(* PLC project Система умного дома.project, CODESYS CODESYS V3.5 SP17 Patch 3 *)
(* stored: creationDateTime 2026-04-06T20:38:17.5908527, modificationDateTime 2026-03-25T09:46:39.3897592 *)

{attribute 'qualified_only'}
{attribute 'strict'}
TYPE E_ALERT_PRIORITY : (ALERT_PRIORITY_NONE := 0, ALERT_PRIORITY_LOW := 1, ALERT_PRIORITY_MEDIUM := 2, ALERT_PRIORITY_HIGH := 3, ALERT_PRIORITY_CRITICAL := 4) BYTE;
END_TYPE

{attribute 'qualified_only'}
{attribute 'strict'}
TYPE E_Debug_Log_Level : (LOG_LEVEL_MINIMAL := 0, LOG_LEVEL_NORMAL := 1, LOG_LEVEL_VERBOSE := 2, LOG_LEVEL_DEBUG := 3) BYTE;
END_TYPE

{attribute 'qualified_only'}
{attribute 'strict'}
TYPE E_Lifetime_Device_Type : (LIFETIME_DEVICE_PUMP := 1, LIFETIME_DEVICE_FAN := 2) BYTE;
END_TYPE

{attribute 'qualified_only'}
{attribute 'strict'}
TYPE E_Outdoor_Mode : (OUTDOOR_MODE_AUTO := 0, OUTDOOR_MODE_PARTY := 1, OUTDOOR_MODE_SECURITY := 2, OUTDOOR_MODE_ECONOMY := 3, OUTDOOR_MODE_MANUAL := 4) BYTE;
END_TYPE

{attribute 'qualified_only'}
{attribute 'strict'}
TYPE E_PLC_ROLE : (ROLE_UNDEFINED := 0, ROLE_ACTIVE := 1, ROLE_STANDBY := 2, ROLE_OFFLINE := 3) USINT;
END_TYPE

{attribute 'qualified_only'}
{attribute 'strict'}
TYPE E_Rule_Action_Type : (ACTION_NONE := 0, ACTION_SET_FLOOR_HEATING := 1, ACTION_SET_LIGHTING_BASE := 2, ACTION_SET_LIGHTING_ACCENT := 3, ACTION_SET_SOCKET := 4, ACTION_SET_VENTILATION := 5, ACTION_SET_BLINDS := 6, ACTION_ACTIVATE_SCENARIO := 7, ACTION_TOGGLE_LIGHTING := 8, ACTION_TOGGLE_SOCKET := 9) BYTE;
END_TYPE

{attribute 'qualified_only'}
{attribute 'strict'}
TYPE E_Rule_Comparison : (COMP_NONE := 0, COMP_EQ := 1, COMP_GT := 2, COMP_LT := 3, COMP_GE := 4, COMP_LE := 5, COMP_IN_RANGE := 6, COMP_TRUE := 7, COMP_FALSE := 8) BYTE;
END_TYPE

(* values of E_Rule_Condition_Type: COND_AND: Логическое И (Rule Chaining); COND_OR: Логическое ИЛИ (Rule Chaining) *)

{attribute 'qualified_only'}
{attribute 'strict'}
TYPE E_Rule_Condition_Type : (COND_NONE := 0, COND_AIR_TEMP := 1, COND_FLOOR_TEMP := 2, COND_HUMIDITY := 3, COND_CO2 := 4, COND_METHANE := 5, COND_CO := 6, COND_DOOR_WINDOW := 7, COND_FLOOD := 8, COND_SMOKE := 9, COND_MOTION := 10, COND_TIME_OF_DAY := 11, COND_DAY_OF_WEEK := 12, COND_AND := 13, COND_OR := 14) BYTE;
END_TYPE

{attribute 'qualified_only'}
{attribute 'strict'}
TYPE E_SCENARIO_TYPE : (SCENARIO_NONE := 0, SCENARIO_MORNING := 1, SCENARIO_EVENING := 2, SCENARIO_AWAY := 3, SCENARIO_PARTY := 4, SCENARIO_SLEEP := 5, SCENARIO_EMERGENCY := 6, SCENARIO_PRESENCE := 7) BYTE;
END_TYPE

{attribute 'qualified_only'}
{attribute 'strict'}
TYPE E_SENSOR_TYPE : (SENSOR_TYPE_NONE := 0, SENSOR_TYPE_DOOR_WINDOW := 5, SENSOR_TYPE_GLASS_BREAK := 6, SENSOR_TYPE_FLOOD := 7, SENSOR_TYPE_SMOKE := 8, SENSOR_TYPE_GAS_METHANE := 1, SENSOR_TYPE_GAS_CO := 2, SENSOR_TYPE_TEMP_FLOOR := 3, SENSOR_TYPE_TEMP_AIR := 4) USINT;
END_TYPE

{attribute 'qualified_only'}
{attribute 'strict'}
TYPE E_Trend_Parameter_Type : (TREND_PARAM_NONE := 0, TREND_PARAM_TEMP_AIR := 1, TREND_PARAM_TEMP_FLOOR := 2, TREND_PARAM_PRESSURE := 3, TREND_PARAM_PUMP_CURRENT := 4, TREND_PARAM_GAS_METHANE := 5, TREND_PARAM_GAS_CO := 6) BYTE;
END_TYPE

{attribute 'qualified_only'}
{attribute 'strict'}
TYPE E_TwoFactor_Method : (TF_METHOD_NONE := 0, TF_METHOD_RFID := 1, TF_METHOD_TOTP := 2, TF_METHOD_BOTH := 3) BYTE;
END_TYPE

{attribute 'qualified_only'}
{attribute 'strict'}
TYPE E_Valve_Test_Result : (TEST_RESULT_NONE := 0, TEST_RESULT_PASSED := 1, TEST_RESULT_CURRENT_DEVIATION := 2, TEST_RESULT_TIME_DEVIATION := 3, TEST_RESULT_STALL := 4, TEST_RESULT_LIMIT_SWITCH_FAIL := 5, TEST_RESULT_ABORTED := 6) BYTE;
END_TYPE

(* values of E_VALVE_TYPE: VALVE_NC: Нормально-закрытый; VALVE_NO: Нормально-открытый *)

{attribute 'qualified_only'}
{attribute 'strict'}
TYPE E_VALVE_TYPE : (VALVE_NC := 1, VALVE_NO := 2) USINT;
END_TYPE

{attribute 'qualified_only'}
{attribute 'strict'}
TYPE E_VENTILATION_LOCATION : (VENT_LOCATION_NONE := 0, VENT_LOCATION_BASEMENT_GAME_ROOM := 1, VENT_LOCATION_BASEMENT_GYM := 2, VENT_LOCATION_BASEMENT_BOILER_ROOM := 3, VENT_LOCATION_BATHROOM_1F := 4, VENT_LOCATION_BATHROOM_2F := 5, VENT_LOCATION_MASTER_BATHROOM := 6, VENT_LOCATION_LAUNDRY := 7, VENT_LOCATION_KITCHEN := 8) BYTE;
END_TYPE

{attribute 'qualified_only'}
{attribute 'strict'}
TYPE E_VENTILATION_UNIT_TYPE : (VENTILATION_TYPE_NONE := 0, VENTILATION_TYPE_SUPPLY := 1, VENTILATION_TYPE_EXHAUST := 2) USINT;
END_TYPE

{attribute 'qualified_only'}
{attribute 'strict'}
TYPE E_WEATHER_COMPENSATION_METHOD : (WEATHER_COMP_NONE := 0, WEATHER_COMP_OUTDOOR_RESET := 1) USINT;
END_TYPE

{attribute 'qualified_only'}
{attribute 'strict'}
TYPE E_Zone_Access_Level : (ZONE_ACCESS_NONE := 0, ZONE_ACCESS_VIEW := 1, ZONE_ACCESS_CONTROL := 2, ZONE_ACCESS_CONFIG := 3, ZONE_ACCESS_FULL := 4) BYTE;
END_TYPE

TYPE ST_Astro_Time : STRUCT
  sunrise_ms : UDINT := 0;
  sunset_ms : UDINT := 0;
  is_daylight : BOOL := FALSE;
END_STRUCT;
END_TYPE

TYPE ST_BlackBox_Record : STRUCT
  Timestamp : UDINT;
  Gas_Methane_LEL : REAL;
  Gas_CO_PPM : REAL;
  Flood_Active : BOOL;
  Fire_Active : BOOL;
  Valve_Gas_Status : BYTE;
  Valve_Water_Status : BYTE;
  PLC_Active_ID : BYTE;
END_STRUCT;
END_TYPE

TYPE ST_Boiler_Status : STRUCT
  Active : BOOL;
  Running : BOOL;
  Error : BOOL;
  Power_Percent : REAL;
  Current_Power : REAL;
  Work_Seconds : UDINT;
  Work_Hours : REAL;
  Resource_Percent : REAL := 100;
  Last_Start : DT;
END_STRUCT;
END_TYPE

TYPE ST_Component_Maintenance : STRUCT
  Is_Faulty : BOOL;  (* Устройство неисправно *)
  Is_In_Maintenance : BOOL;  (* Выведено в ремонт вручную *)
  Fallback_Value : REAL;  (* Значение для подстановки (0-100% или температура) *)
  Use_Last_Good_Value : BOOL;  (* Использовать последнее достоверное значение *)
END_STRUCT;
END_TYPE

TYPE ST_Debug_Log_Record : STRUCT
  timestamp_ms : UDINT;
  level : BYTE;  (* E_Debug_Log_Level *)
  source_id : BYTE;
  event_code : WORD;
  value_int : UDINT;
  value_real : REAL;
  text : STRING(80);
  crc32 : DWORD;
END_STRUCT;
END_TYPE

TYPE ST_Debug_Logger_Config : STRUCT
  enabled : BOOL;
  sampling_period_ms : UDINT := 1000;
END_STRUCT;
END_TYPE

TYPE ST_Device_Health : STRUCT
  Health_Score : BYTE := 100;  (* 0..100% *)
  Total_Runtime_Hours : UDINT;
  Starts_Count : UDINT;
  Last_Start_Current : REAL;
  Avg_Start_Current : REAL;
  Maintenance_Required : BOOL;
  Warning_Message : STRING(50);
END_STRUCT;
END_TYPE

TYPE ST_DHW_Config : STRUCT
  Target_Temp : REAL := 55;
  Hysteresis : REAL := 2;
  Circulation_Schedule_Enabled : BOOL := TRUE;
  Circulation_Start : TOD := TIME_OF_DAY#6:0;
  Circulation_End : TOD := TIME_OF_DAY#23:0;
  Anti_Legionella_Enabled : BOOL := TRUE;
  Anti_Legionella_Day : UINT := 7;  (* Воскресенье *)
END_STRUCT;
END_TYPE

TYPE ST_DHW_Status : STRUCT
  Temp : REAL;
  Pressure : REAL;
  Heating_Pump_On : BOOL;
  Circ_Pump_On : BOOL;
  Error : BOOL;
  Error_ID : WORD;
END_STRUCT;
END_TYPE

TYPE ST_Flood_Config : STRUCT
  Emergency_Two_Stage_Enabled : BOOL := TRUE;  (* ТЗ 4.4 *)
  Valve_Test_Period_Days : UINT := 7;  (* ТЗ 12.2 *)
  Current_Threshold_MA : REAL := 500;  (* Порог тока для диагностики *)
END_STRUCT;
END_TYPE

TYPE ST_Flood_Global_Config : STRUCT
  valve_types : ARRAY[1..3] OF E_VALVE_TYPE := [3(E_VALVE_TYPE.VALVE_NC)];
  min_duration_ms : UDINT := 30000;
END_STRUCT;
END_TYPE

TYPE ST_FloorHeating_Circuit_Config : STRUCT
  circuit_id : BYTE := 0;
  zone : BYTE := 0;
  design_temp : REAL := 35;
  min_temp : REAL := 20;
  max_temp : REAL := 45;
  pid_kp : REAL := 2;
END_STRUCT;
END_TYPE

TYPE ST_FloorHeating_Global_Config : STRUCT
  enable_floor_heating : BOOL := TRUE;
  anti_freeze_temp : REAL := 7;
  overheat_temp : REAL := 45;
  weather_compensation_enabled : BOOL := TRUE;
  total_circuits : BYTE := 16;
END_STRUCT;
END_TYPE

TYPE ST_FloorHeating_Manifold_Config : STRUCT
  manifold_id : BYTE;
  location : STRING(30);
  nominal_flow : REAL;
  enable_pump : BOOL;
  circuits : ARRAY[1..4] OF ST_FloorHeating_Circuit_Config;
END_STRUCT;
END_TYPE

TYPE ST_Gas_Valve_Configuration : STRUCT
  valve_id : BYTE := 0;
  valve_type : E_VALVE_TYPE := E_VALVE_TYPE.VALVE_NC;
  close_time_seconds : UDINT := 10;
  open_time_seconds : UDINT := 10;
  emergency_open_allowed : BOOL := FALSE;
END_STRUCT;
END_TYPE

TYPE ST_Gateway_Command : STRUCT
  command_id : UDINT;
  timestamp_ms : UDINT;
  operator_id : STRING(10);
  command_type : BYTE;
  target_zone : BYTE;
  target_value : REAL;
  target_on_off : BOOL;
  target_scenario : E_SCENARIO_TYPE;
  target_armed : BOOL;
  crc32 : DWORD;
END_STRUCT;
END_TYPE

TYPE ST_Heating_Config : STRUCT
  Weather_Comp_Enabled : BOOL := TRUE;
  Weather_Coef : REAL := 0.1;
  Freeze_Threshold : REAL := 7;
  Overheat_Threshold : REAL := 45;
  Night_Reduction : REAL := 3;
  Target_Floor_Temp : REAL := 28;
  Target_Room_Temp : REAL := 22;
  Hysteresis : REAL := 0.5;
END_STRUCT;
END_TYPE

TYPE ST_History_Record : STRUCT
  timestamp_ms : UDINT := 0;
  event_code : WORD := 0;
  event_value : REAL := 0;
  unit : BYTE := 0;
  zone_id : BYTE := 0;
  operator_id : STRING(10) := '';
  priority : E_ALERT_PRIORITY := E_ALERT_PRIORITY.ALERT_PRIORITY_NONE;
END_STRUCT;
END_TYPE

TYPE ST_Lifetime_Status : STRUCT
  device_id : BYTE;
  runtime_hours : UDINT;
  start_count : UDINT;
  remaining_hours : UDINT;
  remaining_percent : BYTE;
  maintenance_required : BOOL;
  last_calc_timestamp : UDINT;
END_STRUCT;
END_TYPE

TYPE ST_Maintenance_Access_Config : STRUCT
  maintenance_enabled : BOOL := FALSE;
  max_duration_minutes : UDINT := 60;
  requires_two_person : BOOL := TRUE;
  access_level_required : BYTE := 2;
END_STRUCT;
END_TYPE

TYPE ST_Manifold_Status : STRUCT
  Pump_On : BOOL;
  Pump_Current : REAL;
  Pressure : REAL;
  Temp_Supply : REAL;
  Temp_Return : REAL;
  Valve_Pos : REAL;  (* 0-100% *)
  Error : BOOL;
  Error_ID : WORD;
END_STRUCT;
END_TYPE

TYPE ST_Operator_Zone_Rights : STRUCT
  operator_id : STRING(10);
  global_access_level : BYTE := 0;
  zone_masks : ARRAY[1..18] OF DWORD;
  last_modified : UDINT;
END_STRUCT;
END_TYPE

TYPE ST_Outdoor_Zone_Config : STRUCT
  zone_id : BYTE := 0;
  lighting_circuit_id : BYTE := 0;
  auto_enabled : BOOL := TRUE;
  party_mode_enabled : BOOL := FALSE;
END_STRUCT;
END_TYPE

TYPE ST_Owen_Analog_Value : STRUCT
  rValue : REAL;  (* Измеренное значение *)
  uiCycleTime : UINT;  (* Циклическое время *)
  wStatus : WORD;  (* Код статуса (ANALOG_SENSOR_ERRORS) *)
END_STRUCT;
END_TYPE

TYPE ST_Rule_Action : STRUCT
  Active : BOOL;
  Target_ID : BYTE;
  Value : REAL;
END_STRUCT;
END_TYPE

TYPE ST_Scenario_Config : STRUCT
  scenario_id : E_SCENARIO_TYPE;
  lighting_level_base : BYTE := 100;
  lighting_level_accent : BYTE := 100;
  floor_heating_adjust_celsius : REAL := 0;
  ventilation_speed_percent : BYTE := 50;
  sockets_enabled : BOOL := TRUE;
  blinds_position_percent : BYTE := 0;
END_STRUCT;
END_TYPE

TYPE ST_Scenario_Transition_Config : STRUCT
  current_scenario : E_SCENARIO_TYPE;
  target_scenario : E_SCENARIO_TYPE;
  min_duration_minutes : UDINT := 5;
  transition_allowed : BOOL := FALSE;
END_STRUCT;
END_TYPE

TYPE ST_Security_Config : STRUCT
  PIN_Code : STRING(4) := '1234';
  Max_Attempts : UINT := 3;
  Entry_Delay_S : UINT := 45;
  Two_Factor_Enabled : BOOL := FALSE;
  Two_Stage_Mode : BOOL := TRUE;  (* ТЗ 3.4 *)
  Confirmation_Timeout_S : UINT := 120;  (* ТЗ 3.4 (60-300с) *)
  Phones : ARRAY[1..5] OF STRING(15);
  gate_open_pulse_ms : UDINT := 1000;  (* Управление доступом *)
  wicket_open_pulse_ms : UDINT := 1000;
  lock_open_pulse_ms : UDINT := 1000;
  lock_close_pulse_ms : UDINT := 1000;
END_STRUCT;
END_TYPE

TYPE ST_Security_Global_Config : STRUCT
  entry_delay_seconds : UDINT := 30;
  exit_delay_seconds : UDINT := 60;
  alarm_duration_seconds : UDINT := 180;
  two_person_timeout_seconds : UDINT := 120;
  max_access_attempts : BYTE := 3;
  auto_arm_enabled : BOOL := FALSE;
  auto_arm_time_ms : UDINT := 0;
  gate_open_pulse_ms : UDINT := 1000;  (* ТЗ: Управление доступом *)
  wicket_open_pulse_ms : UDINT := 1000;
  lock_open_pulse_ms : UDINT := 1000;
  lock_close_pulse_ms : UDINT := 1000;
END_STRUCT;
END_TYPE

TYPE ST_Security_Zone_State : STRUCT
  Armed : BOOL;
  Alarm : BOOL;
  Bypassed : BOOL;
  Last_Trigger_Time : DT;
  Trigger_Count : UINT;
END_STRUCT;
END_TYPE

TYPE ST_Sensor_Calibration_Record : STRUCT
  sensor_id : UDINT := 0;
  sensor_type : E_SENSOR_TYPE;
  zone_id : BYTE := 0;
  offset : REAL := 0;
  multiplier : REAL := 1;
  last_calibration_timestamp : UDINT := 0;
  verification_passed : BOOL := FALSE;
END_STRUCT;
END_TYPE

TYPE ST_State_Snapshot : STRUCT
  timestamp_ms : UDINT := 0;
  operator_id : STRING(10) := '';
  scenario_id : E_SCENARIO_TYPE := E_SCENARIO_TYPE.SCENARIO_NONE;
  lighting_levels : ARRAY[1..16] OF BYTE;
  floor_heating_setpoints : ARRAY[1..16] OF REAL;
  alarm_active : BOOL := FALSE;
  crc32 : DWORD := 0;
END_STRUCT;
END_TYPE

TYPE ST_System_State_Summary : STRUCT
  Outdoor_Temp : REAL;
  Indoor_Temp : ARRAY[1..16] OF REAL;
  Floor_Temps : ARRAY[1..16] OF REAL;
  Humidity : ARRAY[1..8] OF REAL;
  CO2 : ARRAY[1..8] OF REAL;
  Gas_Alarm : BOOL;
  Flood_Alarm : BOOL;
  Fire_Alarm : BOOL;
  Security_Armed : BOOL;
END_STRUCT;
END_TYPE

TYPE ST_Tariff_Config : STRUCT
  Enabled : BOOL := FALSE;
  Night_Start_Hour : UINT := 23;  (* 23:00 *)
  Night_End_Hour : UINT := 7;  (* 07:00 *)
  Boost_Delta : REAL := 2;  (* На сколько градусов поднять уставку ночью *)
END_STRUCT;
END_TYPE

TYPE ST_Trend_Config : STRUCT
  param_type : BYTE;  (* E_Trend_Parameter_Type *)
  zone_id : BYTE;
  enabled : BOOL;
  deviation_threshold_percent : REAL := 10;
  history_days : UDINT := 7;
END_STRUCT;
END_TYPE

TYPE ST_Trend_Data : STRUCT
  config : ST_Trend_Config;
  record_count : UDINT;
  write_index : UDINT;
  sum_values : REAL;
  crc32 : DWORD;
END_STRUCT;
END_TYPE

TYPE ST_Trend_Header : STRUCT
  parameter_type : BYTE;  (* E_Trend_Parameter_Type *)
  zone_id : BYTE := 0;
  records_count : UDINT := 0;
  average_value : REAL := 0;
  min_value : REAL := 0;
  max_value : REAL := 0;
END_STRUCT;
END_TYPE

TYPE ST_Trend_History_Record : STRUCT
  timestamp_ms : UDINT := 0;
  value : REAL := 0;
END_STRUCT;
END_TYPE

TYPE ST_TwoFactor_Auth_State : STRUCT
  operator_id : STRING(10);
  is_pending : BOOL;  (* Ожидание ввода 2-го фактора *)
  start_time : UDINT;
  timeout_ms : UDINT := 60000;
END_STRUCT;
END_TYPE

TYPE ST_TwoFactor_Data : STRUCT
  operator_id : STRING(10);
  AuthMethod : BYTE;  (* E_TwoFactor_Method *)
  rfid_tag : STRING(20);
  totp_secret : STRING(32);
  last_modified : UDINT;
END_STRUCT;
END_TYPE

TYPE ST_User_Rule : STRUCT
  Enabled : BOOL;
  Condition_Type : BYTE;  (* 1-Temp, 2-Hum, 3-CO2, 4-Security, 5-Time *)
  Condition_Op : BYTE;  (* 1:>, 2:<, 3:= *)
  Condition_Value : REAL;
  Action_Target_ID : BYTE;
  Action_Value : REAL;
  Action_Type : BYTE;  (* 1-SetTemp, 2-Switch, 3-Scenario *)
  Priority : BYTE;  (* ТЗ 7.4: Приоритет (0-255) *)
END_STRUCT;
END_TYPE

TYPE ST_Valve_Test_Config : STRUCT
  valve_id : BYTE := 0;
  test_interval_days : UDINT := 7;
  nominal_current_a : REAL := 0.5;
  Nominal_Current : REAL := 0.5;
  nominal_close_time_sec : REAL := 10;
  enabled : BOOL := TRUE;
END_STRUCT;
END_TYPE

TYPE ST_Ventilation_Config : STRUCT
  CO2_Threshold : REAL := 800;
  Humidity_Threshold : REAL := 65;
  Night_Mode_Start : TOD := TIME_OF_DAY#23:0;
  Night_Mode_End : TOD := TIME_OF_DAY#7:0;
END_STRUCT;
END_TYPE

TYPE ST_Ventilation_Global_Config : STRUCT
  enable_ventilation : BOOL := TRUE;
  total_units : BYTE := 8;
  default_supply_speed : BYTE := 40;
  default_exhaust_speed : BYTE := 40;
END_STRUCT;
END_TYPE

TYPE ST_Ventilation_Scenario_Mode : STRUCT
  Scenario_ID : BYTE;
  Scenario_Priority : BYTE;
  Fire_Alarm : BOOL;
  Methane_Alarm : BOOL;
  Smoke_Detected : BOOL;
  Exhaust_Modes : ARRAY[1..5] OF BYTE;
  Supply_Modes : ARRAY[1..3] OF BYTE;
END_STRUCT;
END_TYPE

TYPE ST_Ventilation_Unit : STRUCT
  Enabled : BOOL;
  Speed_Percent : REAL;
  Filter_Dirty : BOOL;
  Error : BOOL;
  Mode : BYTE;  (* 0-Eco, 1-Std, 2-Int, 3-Emergency *)
END_STRUCT;
END_TYPE

TYPE ST_Ventilation_Unit_Config : STRUCT
  unit_id : BYTE := 0;
  unit_type : E_VENTILATION_UNIT_TYPE;
  location : E_VENTILATION_LOCATION;
  min_speed : BYTE := 20;
  max_speed : BYTE := 100;
  Threshold_Hum : REAL := 65;
  has_smoke_detector : BOOL := FALSE;
END_STRUCT;
END_TYPE

TYPE ST_Zone_Sensors : STRUCT
  Temp_Room : REAL;
  Temp_Floor : REAL;
  Motion_Active : BOOL;
  Switch_Physical : BOOL;
  Light_State : BOOL;
  Maintenance : ST_Component_Maintenance;
END_STRUCT;
END_TYPE

{attribute 'qualified_only'}
VAR_GLOBAL  (* GVL_BlackBox *)
  G_BlackBox_Buffer : ARRAY[0..99] OF ST_BlackBox_Record;  (* Буфер на 100 записей (при опросе 100мс это 10 секунд истории) *)
  G_BlackBox_Frozen : BOOL;
  G_BlackBox_LastIndex : INT;
END_VAR

{attribute 'qualified_only'}
VAR_GLOBAL CONSTANT  (* GVL_Constants *)
  C_MS_PER_SEC : UDINT := 1000;
  C_SEC_PER_MIN : UDINT := 60;
  C_MIN_PER_HOUR : UDINT := 60;
  C_MS_PER_MIN : UDINT := 60000;
  C_MAX_RULES : INT := 20;
  C_ZONE_COUNT : BYTE := 18;
END_VAR

{attribute 'qualified_only'}
VAR_GLOBAL  (* GVL_Diagnostics *)
  G_Pump_Health : ARRAY[1..5] OF ST_Device_Health;  (* Для 5 коллекторных насосов *)
  G_Gas_Valve_Health : ST_Device_Health;
  G_System_Health_Summary : BYTE := 100;
END_VAR

{attribute 'qualified_only'}
VAR_GLOBAL  (* GVL_Global_Variables *)
  GVL_System_Time_MS : UDINT;
  GVL_IsActivePLC : BOOL := TRUE;
  GVL_Local_PLC_Role : E_PLC_ROLE := E_PLC_ROLE.ROLE_ACTIVE;
  GVL_Floor_Temps : ARRAY[1..16] OF REAL;  (* Данные датчиков *)
  GVL_Valve_States : ARRAY[1..3] OF BYTE;
END_VAR

VAR_GLOBAL  (* GVL_HMI_Config *)
  G_HMI_FloorHeating_Configs : ARRAY[1..16] OF ST_FloorHeating_Circuit_Config;  (* Настройки отопления (16 контуров) *)
  G_HMI_Tariff_Settings : ST_Tariff_Config;
  G_HMI_Vent_Global_Config : ST_Ventilation_Global_Config;  (* Настройки вентиляции (8 установок) *)
  G_HMI_Vent_Unit_Configs : ARRAY[1..8] OF ST_Ventilation_Unit_Config;
  G_HMI_Scenario_Configs : ARRAY[1..6] OF ST_Scenario_Config;  (* Для каждого типа сценария *)
  G_HMI_Outdoor_Configs : ARRAY[1..4] OF ST_Outdoor_Zone_Config;
  G_HMI_Flood_Config : ST_Flood_Global_Config;  (* Настройки безопасности *)
  G_HMI_Cleaning_Mode_Active : ARRAY[1..3] OF BOOL;  (* Режим уборки для 3-х зон протечки *)
  G_HMI_Cleaning_Mode_TimeLeft : ARRAY[1..3] OF UINT;  (* Оставшееся время (мин) *)
  G_HMI_Gas_Config : ST_Gas_Valve_Configuration;
  G_HMI_Admin_2FA_Enabled : BOOL := FALSE;  (* Настройка: 1 или 2 фактора для ADMIN *)
  G_HMI_Current_Operator_Factor2_Done : BOOL;  (* Флаг прохождения 2-го фактора *)
  G_HMI_Sensor_Calibrations : ARRAY[1..20] OF ST_Sensor_Calibration_Record;  (* Калибровка датчиков (например, для 20 датчиков) *)
  G_HMI_Current_Operator_ID : STRING(10);  (* ID текущего авторизованного пользователя *)
  G_HMI_Manual_Gas_Valve_Open : BOOL;  (* Запрос на открытие *)
  G_HMI_Manual_Gas_Valve_Time : UDINT := 5;  (* Время в минутах *)
  G_HMI_Manual_Gas_Valve_TimeLeft : UDINT;  (* Оставшееся время (для вывода на HMI) *)
  G_HMI_Apply_Settings : BOOL;  (* Команда на сохранение настроек в NVRAM *)
  G_HMI_Gate_Open_Req : BOOL;  (* Управление доступом (HMI) *)
  G_HMI_Wicket_Open_Req : BOOL;
  G_HMI_Lock_1_Open_Req : BOOL;
  G_HMI_Lock_1_Close_Req : BOOL;
  G_HMI_Lock_2_Open_Req : BOOL;
  G_HMI_Lock_2_Close_Req : BOOL;
END_VAR

VAR_GLOBAL  (* GVL_IO *)
  DI_Security_Open : ARRAY[1..15] OF BOOL;  (* Датчики открытия (15 физических каналов по ТЗ 3.1) *)
  DI_Security_Glass : ARRAY[1..15] OF BOOL;  (* Датчики разбития (15 физических каналов по ТЗ 3.2) *)
  DI_Security_2F_Group : BOOL;  (* Групповой канал 2-го этажа *)
  DI_Flood_Sensors : ARRAY[1..12] OF BOOL;  (* Датчики протечки (12 штук по ТЗ 4.1) *)
  AO_Manifold_Valves : ARRAY[1..5] OF UINT;  (* 0-1000 (Modbus) *)
  DO_Manifold_Pumps : ARRAY[1..5] OF BOOL;
  AI_Manifold_Currents : ARRAY[1..5] OF INT;  (* 4-20mA -> 400-2000 *)
  AI_Manifold_Pressures : ARRAY[1..5] OF INT;  (* 0-10V -> 0-1000 *)
  AI_Manifold_Temps_Supply : ARRAY[1..5] OF ST_Owen_Analog_Value;
  AI_Manifold_Temps_Return : ARRAY[1..5] OF INT;
  AO_Supply_Fans : ARRAY[1..3] OF UINT;  (* 0-1000 *)
  AO_Exhaust_Fans : ARRAY[1..5] OF UINT;  (* 0-1000 *)
  DO_Boiler_Enable : ARRAY[1..2] OF BOOL;  (* Котлы (BAXI Luna Platinum+ через OpenTherm) *)
  AO_Boiler_Setpoint : ARRAY[1..2] OF UINT;  (* 0-1000 (0-100.0 C) *)
  AI_Boiler_Modulation : ARRAY[1..2] OF INT;
  AI_Boiler_Flame_Status : ARRAY[1..2] OF BOOL;
  DI_Boiler_Error : ARRAY[1..2] OF BOOL;
  AI_Methane_LEL : ARRAY[1..2] OF ST_Owen_Analog_Value;  (* 0-100% LEL *)
  AI_CO_PPM : ARRAY[1..8] OF REAL;  (* 0-1000 PPM *)
  DI_Smoke_Sensors : ARRAY[1..6] OF BOOL;
  AI_Temp_Outdoor : ST_Owen_Analog_Value;  (* Аналоговые входы (AI) *)
  AI_Floor_Temps : ARRAY[1..16] OF REAL;
  AI_Room_Temps : ARRAY[1..16] OF REAL;  (* Датчики температуры помещения (ТЗ 1.1) *)
  DO_Zone_Valves : ARRAY[1..16] OF BOOL;  (* Клапаны контуров ТП *)
  AI_DHW_Temp : REAL;  (* ГВС (ТЗ 5.0) *)
  AI_DHW_Pressure : REAL;
  DO_DHW_Heating_Pump : BOOL;
  DO_DHW_Circ_Pump : BOOL;
  DI_Lighting_Switches : ARRAY[1..16] OF BOOL;  (* Освещение и Движение (ТЗ 1.0, 2.0) *)
  DI_Motion_Sensors : ARRAY[1..16] OF BOOL;
  DO_Gas_Valve_Close : BOOL;  (* Безопасность и Аварии *)
  DO_Water_Valve_35_Close : BOOL;
  DO_Water_Valve_36_Close : BOOL;
  AI_Water_Valve_35_Current : REAL;
  AI_Water_Valve_36_Current : REAL;
  DI_Power_OK : BOOL;
  DO_Gas_Siren : BOOL;
  DO_Fire_Siren : BOOL;
  DO_Pump_Main_Enable : BOOL;
  DO_Gate_Open : BOOL;  (* Управление доступом (Сухие контакты) *)
  DO_Wicket_Open : BOOL;
  DO_Lock_1_Open : BOOL;
  DO_Lock_1_Close : BOOL;
  DO_Lock_2_Open : BOOL;
  DO_Lock_2_Close : BOOL;
END_VAR

VAR_GLOBAL  (* GVL_Vars *)
  G_System_Time_MS : UDINT;  (* Системное время (мс) *)
  G_Current_Scenario : E_SCENARIO_TYPE := E_SCENARIO_TYPE.SCENARIO_NONE;
  G_Security_Armed : BOOL := FALSE;
  G_Gas_Alarm_Active : BOOL := FALSE;
  G_Fire_Alarm_Active : BOOL := FALSE;
  G_Flood_Alarm_Active : BOOL := FALSE;
  G_Local_PLC_ID : BYTE := 1;  (* ID текущего ПЛК (1 для A, 2 для B) *)
  G_Active_PLC_ID : BYTE := 1;  (* ID активного ПЛК в данный момент *)
  G_Remote_PLC_Pulse : BOOL;  (* Импульс от партнера *)
  G_HMI_Current_Operator_ID : STRING(10) := 'ADMIN';  (* HMI и Конфигурация *)
  G_HMI_Gas_Config : ST_Gas_Valve_Configuration;
  G_Heating_Config : ST_Heating_Config;
  G_Ventilation_Config : ST_Ventilation_Config;
  G_DHW_Config : ST_DHW_Config;
  G_Security_Config : ST_Security_Config;
  G_Flood_Config : ST_Flood_Config;
  G_HMI_Mute_Alarm : BOOL;
  G_HMI_Manual_Gas_Valve_Open : BOOL;
  G_HMI_Manual_Gas_Valve_Time : UDINT := 300000;  (* 5 минут по умолчанию *)
  G_HMI_Manual_Gas_Valve_TimeLeft : UDINT;
  G_Floor_Temps : ARRAY[1..16] OF REAL;  (* Состояние датчиков *)
  G_BlackBox_Buffer : ARRAY[0..99] OF ST_BlackBox_Record;  (* Черный ящик *)
  G_BlackBox_LastIndex : INT;
  G_BlackBox_Frozen : BOOL;
  G_Maintenance_Zones : ARRAY[1..16] OF ST_Component_Maintenance;  (* ТЗ 6.0: Обслуживание и ремонт *)
  G_Maintenance_Manifolds : ARRAY[1..5] OF ST_Component_Maintenance;
  G_Maintenance_Lighting : ARRAY[1..16] OF ST_Component_Maintenance;
  G_HMI_Gate_Open_Req : BOOL;  (* Управление доступом (HMI) *)
  G_HMI_Wicket_Open_Req : BOOL;
  G_HMI_Lock_1_Open_Req : BOOL;
  G_HMI_Lock_1_Close_Req : BOOL;
  G_HMI_Lock_2_Open_Req : BOOL;
  G_HMI_Lock_2_Close_Req : BOOL;
END_VAR

INTERFACE IValveController
METHOD OpenValve : BOOL
  VAR_INPUT
    VI_Operator_ID : STRING(10);
    VI_Force : BOOL;
  END_VAR
END_METHOD
METHOD CloseValve : BOOL
  VAR_INPUT
    VI_Operator_ID : STRING(10);
    VI_Force : BOOL;
  END_VAR
END_METHOD
METHOD GetStatus : BYTE
END_METHOD
END_INTERFACE

PROGRAM PRG_PLC_A
  VAR
    L_PLC_ID : BYTE := 1;
  END_VAR

            // Вызов основной программы
PRG_System();
// >>> BULK_SYNC_ANCHOR: PRG_PLC_A <<<

          
END_PROGRAM

PROGRAM PRG_PLC_B
  VAR
    L_PLC_ID : BYTE := 2;
  END_VAR

            // Вызов основной программы
PRG_System();
// >>> BULK_SYNC_ANCHOR: PRG_PLC_B <<<

          
END_PROGRAM

FUNCTION_BLOCK FB_Access_Control
  VAR_INPUT
    VI_System_Time_MS : UDINT;
    VI_IsActivePLC : BOOL;
    VI_Armed : BOOL;  (* Состояние охраны *)
    VI_Gate_Open_Req : BOOL;  (* Команды HMI *)
    VI_Wicket_Open_Req : BOOL;
    VI_Lock_1_Open_Req : BOOL;
    VI_Lock_1_Close_Req : BOOL;
    VI_Lock_2_Open_Req : BOOL;
    VI_Lock_2_Close_Req : BOOL;
    VI_Config : ST_Security_Config;  (* Настройки *)
  END_VAR
  VAR_OUTPUT
    VO_Gate_Open : BOOL;
    VO_Wicket_Open : BOOL;
    VO_Lock_1_Open : BOOL;
    VO_Lock_1_Close : BOOL;
    VO_Lock_2_Open : BOOL;
    VO_Lock_2_Close : BOOL;
  END_VAR
  VAR
    L_Gate_Timer : TON;
    L_Wicket_Timer : TON;
    L_Lock_1_Open_T : TON;
    L_Lock_1_Close_T : TON;
    L_Lock_2_Open_T : TON;
    L_Lock_2_Close_T : TON;
    L_Prev_Armed : BOOL;
    L_Auto_Lock_Req : BOOL;
  END_VAR

            // Если ПЛК находится в режиме Standby (резерв), он не должен управлять выходами
IF NOT VI_IsActivePLC THEN
    RETURN;
END_IF;

IF VI_System_Mode = E_System_Operating_Mode.MODE_SAFE_STOP THEN
    VO_Gate_Open := FALSE;
    VO_Wicket_Open := FALSE;
    VO_Lock_1_Open := FALSE;
    VO_Lock_2_Open := FALSE;
    RETURN;
END_IF;

// 1. Логика автоматического закрытия замков при постановке на охрану (ТЗ 3.0)
// При переходе системы в режим "Охрана" принудительно блокируем все замки
IF VI_Armed AND NOT L_Prev_Armed THEN
    L_Auto_Lock_Req := TRUE;
END_IF;
L_Prev_Armed := VI_Armed;

// Детекторы фронта для команд
R_Trig_Gate(CLK := VI_Gate_Open_Req);
R_Trig_Wicket(CLK := VI_Wicket_Open_Req);
R_Trig_Lock_1_O(CLK := VI_Lock_1_Open_Req);
R_Trig_Lock_1_C(CLK := VI_Lock_1_Close_Req OR L_Auto_Lock_Req);
R_Trig_Lock_2_O(CLK := VI_Lock_2_Open_Req);
R_Trig_Lock_2_C(CLK := VI_Lock_2_Close_Req OR L_Auto_Lock_Req);

// Проверка PIN-кода или RFID-метки через менеджер кодов
fbAccessCode(
    VI_System_Time_MS := VI_System_Time_MS,
    VI_IsActivePLC := VI_IsActivePLC,
    VI_Code_To_Check := VI_PIN_Code,
    VI_RFID_To_Check := VI_RFID_Tag,
    VI_Access_Codes := VI_Access_Codes,
    VI_RFID_Tags := VI_RFID_Tags,
    VO_Code_Valid => L_Valid_PIN
);

// 2. Формирование импульсов управления исполнительными механизмами (Pulse Control)
// Открытие ворот и калитки требует валидного ПИН-кода или RFID-метки, если система под охраной
L_Gate_Timer(IN := R_Trig_Gate.Q AND (NOT VI_Armed OR L_Valid_PIN), PT := TO_TIME(VI_Config.gate_open_pulse_ms));
VO_Gate_Open := L_Gate_Timer.Q;

L_Wicket_Timer(IN := R_Trig_Wicket.Q AND (NOT VI_Armed OR L_Valid_PIN), PT := TO_TIME(VI_Config.wicket_open_pulse_ms));
VO_Wicket_Open := L_Wicket_Timer.Q;

L_Lock_1_Open_T(IN := R_Trig_Lock_1_O.Q AND (NOT VI_Armed OR L_Valid_PIN), PT := TO_TIME(VI_Config.lock_open_pulse_ms));
VO_Lock_1_Open := L_Lock_1_Open_T.Q;

L_Lock_1_Close_T(IN := R_Trig_Lock_1_C.Q, PT := TO_TIME(VI_Config.lock_close_pulse_ms));
VO_Lock_1_Close := L_Lock_1_Close_T.Q;

L_Lock_2_Open_T(IN := R_Trig_Lock_2_O.Q AND (NOT VI_Armed OR L_Valid_PIN), PT := TO_TIME(VI_Config.lock_open_pulse_ms));
VO_Lock_2_Open := L_Lock_2_Open_T.Q;

L_Lock_2_Close_T(IN := R_Trig_Lock_2_C.Q, PT := TO_TIME(VI_Config.lock_close_pulse_ms));
VO_Lock_2_Close := L_Lock_2_Close_T.Q;

// Сброс флага автоматического закрытия
IF L_Auto_Lock_Req THEN
    L_Auto_Lock_Req := FALSE;
END_IF;
// >>> BULK_SYNC_ANCHOR: FB_Access_Control <<<

          
END_FUNCTION_BLOCK

FUNCTION_BLOCK FB_AccessCode_Manager
  VAR_INPUT
    VI_System_Time_MS : UDINT;
    VI_IsActivePLC : BOOL;
    VI_Code_To_Check : STRING(4);
  END_VAR
  VAR_OUTPUT
    VO_Code_Valid : BOOL;
  END_VAR
  VAR
    L_Codes : ARRAY[1..5] OF STRING(4) := ['1234', '5678', '0000', '1111', '2222'];
    L_i : INT;
  END_VAR

            VO_Code_Valid := FALSE;

// Вычисляем хэш введенного кода
IF LEN(VI_Code_To_Check) > 0 THEN
    pCode := ADR(VI_Code_To_Check);
    L_Input_Hash := L_CRC_Calc.Calculate(VI_DataRef := pCode^, VI_Size := TO_UDINT(LEN(VI_Code_To_Check)));
    FOR L_i := 1 TO GVL_CONSTANTS.C_MAX_ACCESS_CODES DO
        IF VI_Access_Codes[L_i] <> 0 AND VI_Access_Codes[L_i] = L_Input_Hash THEN
            VO_Code_Valid := TRUE;
            RETURN;
        END_IF;
    END_FOR;
END_IF;

// Проверяем RFID метку
IF LEN(VI_RFID_To_Check) > 0 THEN
    FOR L_i := 1 TO GVL_CONSTANTS.C_MAX_ACCESS_CODES DO
        IF VI_RFID_Tags[L_i] <> '' AND VI_RFID_Tags[L_i] = VI_RFID_To_Check THEN
            VO_Code_Valid := TRUE;
            RETURN;
        END_IF;
    END_FOR;
END_IF;
// >>> BULK_SYNC_ANCHOR: FB_AccessCode_Manager <<<

          
END_FUNCTION_BLOCK

FUNCTION_BLOCK FB_Astro_Timer
  VAR_INPUT
    VI_System_Time_MS : UDINT;
    VI_Latitude : REAL := 55.75;  (* Москва *)
    VI_Longitude : REAL := 37.61;
  END_VAR
  VAR_OUTPUT
    VO_Sunset_Time : TOD;
    VO_Sunrise_Time : TOD;
    VO_Is_Night : BOOL;
  END_VAR
  VAR
    L_Current_TOD : TOD;
  END_VAR

            L_Current_TOD := GVL_STATUS.G_Current_TOD;
VO_Current_TOD := L_Current_TOD;

// Equation of Time (EoT) in minutes
L_B := 360.0 / 365.0 * TO_REAL(VI_Day_Of_Year - 81) * L_Rad;
L_EoT := 9.87 * SIN(2.0 * L_B) - 7.53 * COS(L_B) - 1.5 * SIN(L_B);

// Solar Declination in degrees
L_Declination := 23.45 * SIN(360.0 / 365.0 * TO_REAL(VI_Day_Of_Year + 284) * L_Rad);

// Hour angle
L_Cos_Omega := -TAN(VI_Latitude * L_Rad) * TAN(L_Declination * L_Rad);

IF L_Cos_Omega > 1.0 THEN
    L_Cos_Omega := 1.0; // Polar night
ELSIF L_Cos_Omega < -1.0 THEN
    L_Cos_Omega := -1.0; // Polar day
END_IF;

L_Omega := ACOS(L_Cos_Omega) * L_Deg;

// Sunrise and Sunset in local time (hours)
L_Sunrise_Local := 12.0 - (L_Omega / 15.0) - (L_EoT / 60.0) + (VI_Timezone * 15.0 - VI_Longitude) / 15.0;
L_Sunset_Local := 12.0 + (L_Omega / 15.0) - (L_EoT / 60.0) + (VI_Timezone * 15.0 - VI_Longitude) / 15.0;

// Handle bounds
IF L_Sunrise_Local < 0.0 THEN L_Sunrise_Local := L_Sunrise_Local + 24.0; END_IF;
IF L_Sunrise_Local >= 24.0 THEN L_Sunrise_Local := L_Sunrise_Local - 24.0; END_IF;
IF L_Sunset_Local < 0.0 THEN L_Sunset_Local := L_Sunset_Local + 24.0; END_IF;
IF L_Sunset_Local >= 24.0 THEN L_Sunset_Local := L_Sunset_Local - 24.0; END_IF;

// Конвертация в TOD
VO_Sunrise_Time := TO_TOD(TO_UDINT(L_Sunrise_Local * 3600000.0));
VO_Sunset_Time := TO_TOD(TO_UDINT(L_Sunset_Local * 3600000.0));

// ТЗ 15.2: Закат + 30 мин / Рассвет - 30 мин
VO_Is_Night := (L_Current_TOD > (VO_Sunset_Time + T#30m)) OR (L_Current_TOD < (VO_Sunrise_Time - T#30m));
// >>> SYNC_TEST_MARKER_FORCE <<<
// >>> BULK_SYNC_ANCHOR: FB_Astro_Timer <<<

          
END_FUNCTION_BLOCK

FUNCTION_BLOCK FB_BlackBox_Recorder
  VAR_INPUT
    VI_Current_Data : ST_BlackBox_Record;
    VI_Freeze : BOOL;
  END_VAR
  VAR
    L_Write_Index : INT := 0;
    L_FileHandle : RTS_IEC_HANDLE;
    L_FileName : STRING := '/home/root/blackbox_dump.bin';
    L_FileResult : RTS_IEC_RESULT;
    L_State : INT;
  END_VAR

            IF NOT L_Initialized THEN
    L_Write_Index := GVL_Retain.G_BlackBox_LastIndex;
    IF L_Write_Index < 0 OR L_Write_Index >= GVL_CONSTANTS.C_MAX_BLACKBOX_RECORDS THEN
        L_Write_Index := 0;
        GVL_Retain.G_BlackBox_LastIndex := 0;
    END_IF;
    L_Initialized := TRUE;
END_IF;

IF VI_Freeze THEN
    GVL_Retain.G_BlackBox_Frozen := TRUE;
END_IF;

VO_Frozen := GVL_Retain.G_BlackBox_Frozen;

IF NOT GVL_Retain.G_BlackBox_Frozen THEN
    GVL_Retain.G_BlackBox_Buffer[L_Write_Index] := VI_Current_Data;
    GVL_Retain.G_BlackBox_LastIndex := L_Write_Index;
    
    L_Write_Index := L_Write_Index + 1;
    IF L_Write_Index >= GVL_CONSTANTS.C_MAX_BLACKBOX_RECORDS THEN
        L_Write_Index := 0;
    END_IF;
END_IF;

VO_Records_Count := GVL_CONSTANTS.C_MAX_BLACKBOX_RECORDS; // Размер кольцевого буфера
// >>> BULK_SYNC_ANCHOR: FB_BlackBox_Recorder <<<

          
END_FUNCTION_BLOCK

FUNCTION_BLOCK FB_Boiler_Cascade_Controller
  VAR_INPUT
    VI_Demand_kW : REAL;
    VI_IsActivePLC : BOOL;
  END_VAR
  VAR_OUTPUT
    VO_Boiler1_On : BOOL;
    VO_Boiler2_On : BOOL;
  END_VAR
  VAR
    L_Lead_Boiler : BYTE := 1;  (* 1 или 2 *)
    L_Boiler1_Hours : UDINT;
    L_Boiler2_Hours : UDINT;
    L_Last_Hour_Update : UDINT;
    L_System_Time : UDINT;
  END_VAR
  VAR_INPUT
    VI_System_Time : UDINT;
  END_VAR

            // Логика ротации по наработке
IF (VI_System_Time - L_Last_Hour_Update) >= 3600000 THEN // Раз в час
    L_Last_Hour_Update := VI_System_Time;
    IF VO_Boiler1_On THEN L_Boiler1_Hours := L_Boiler1_Hours + 1; END_IF;
    IF VO_Boiler2_On THEN L_Boiler2_Hours := L_Boiler2_Hours + 1; END_IF;
    
    // Смена ведущего, если разница более 100 часов
    IF (L_Boiler1_Hours > L_Boiler2_Hours + 100) THEN
        L_Lead_Boiler := 2;
    ELSIF (L_Boiler2_Hours > L_Boiler1_Hours + 100) THEN
        L_Lead_Boiler := 1;
    END_IF;
END_IF;

IF VI_IsActivePLC THEN
    IF VI_Demand_kW > 24.0 THEN
        VO_Boiler1_On := TRUE;
        VO_Boiler2_On := TRUE;
    ELSIF VI_Demand_kW > 2.0 THEN
        VO_Boiler1_On := (L_Lead_Boiler = 1);
        VO_Boiler2_On := (L_Lead_Boiler = 2);
    ELSE
        VO_Boiler1_On := FALSE;
        VO_Boiler2_On := FALSE;
    END_IF;
END_IF;

          
END_FUNCTION_BLOCK

FUNCTION_BLOCK FB_Boiler_Cascade_Manager
  VAR_INPUT
    VI_Boiler1_Status : ST_Boiler_Status;
    VI_Boiler2_Status : ST_Boiler_Status;
    VI_Role_Swap_Interval : UDINT := 168;  (* часы *)
  END_VAR
  VAR_OUTPUT
    VO_Boiler1_Enable : BOOL;
    VO_Boiler2_Enable : BOOL;
  END_VAR

            // Логика п. 2.8: Включение резервного при >80% мощности или отказе
IF VI_Boiler1_Status.Error OR VI_Boiler1_Status.Current_Power > 80.0 THEN
    VO_Boiler2_Enable := TRUE;
ELSE
    VO_Boiler2_Enable := FALSE;
END_IF;

VO_Boiler1_Enable := NOT VI_Boiler1_Status.Error;

          
END_FUNCTION_BLOCK

FUNCTION_BLOCK FB_Calibration_Manager
  VAR_INPUT
    VI_Raw_Value : REAL;
    VI_Type : BYTE;  (* 1-Temp, 2-Pressure, 3-Gas *)
    VI_Calib_Record : ST_Sensor_Calibration_Record;
    VI_System_Time_MS : UDINT;
    VI_Start_Verification : BOOL;
  END_VAR
  VAR_OUTPUT
    VO_Calibrated_Value : REAL;
    VO_Verification_Active : BOOL;
    VO_Verification_Failed : BOOL;
    VO_Deviation_Percent : REAL;
  END_VAR
  VAR
    L_Verification_Timer : TON;
    L_Initial_Value : REAL;
  END_VAR

            // 1. Расчет калиброванного значения
CASE VI_Type OF
    1: VO_Calibrated_Value := VI_Raw_Value + VI_Calib_Record.offset;
    2, 3: VO_Calibrated_Value := (VI_Raw_Value * VI_Calib_Record.multiplier) + VI_Calib_Record.offset;
END_CASE;

// 2. Верификация через 1 час (ТЗ 9.5)
IF VI_Start_Verification AND NOT VO_Verification_Active THEN
    VO_Verification_Active := TRUE;
    L_Initial_Value := VO_Calibrated_Value;
    L_Verification_Timer(IN := TRUE, PT := T#1h);
END_IF;

L_Verification_Timer(IN := VO_Verification_Active);

IF L_Verification_Timer.Q THEN
    VO_Verification_Active := FALSE;
    L_Verification_Timer(IN := FALSE);
    
    // ТЗ 9.5: Отклонение ≤2.0% (норма) / >5.0% (ошибка)
    IF L_Initial_Value <> 0 THEN
        VO_Deviation_Percent := ABS(VO_Calibrated_Value - L_Initial_Value) / L_Initial_Value * 100.0;
    ELSE
        VO_Deviation_Percent := 0.0;
    END_IF;
    
    VO_Verification_Failed := (VO_Deviation_Percent > 5.0);
END_IF;

          
END_FUNCTION_BLOCK

FUNCTION_BLOCK FB_CO_Detector
  VAR_INPUT
    VI_CO_PPM : REAL;
    VI_Threshold_Warning : REAL := 30;
    VI_Threshold_Alarm : REAL := 70;
  END_VAR
  VAR_OUTPUT
    VO_Warning_Active : BOOL;
    VO_Alarm_Active : BOOL;
  END_VAR

            VO_Warning_Active := (VI_CO_PPM >= VI_Threshold_Warning);
VO_Alarm_Active := (VI_CO_PPM >= VI_Threshold_Alarm);

          
END_FUNCTION_BLOCK

FUNCTION_BLOCK FB_CRC32_Calculator
  VAR
    L_Table : ARRAY[0..255] OF DWORD;
    L_Initialized : BOOL := FALSE;
    L_i : INT;
    L_j : INT;
    L_Entry : DWORD;
  END_VAR

            
          

METHOD InitTable
                  IF L_Initialized THEN RETURN; END_IF;

FOR L_i := 0 TO 255 DO
    L_Entry := TO_DWORD(L_i);
    FOR L_j := 0 TO 7 DO
        IF (L_Entry AND 1) <> 0 THEN
            L_Entry := SHR(L_Entry, 1) XOR 16#EDB88320;
        ELSE
            L_Entry := SHR(L_Entry, 1);
        END_IF;
    END_FOR;
    L_Table[L_i] := L_Entry;
END_FOR;
L_Initialized := TRUE;
                
END_METHOD

METHOD Calculate : DWORD
  VAR_INPUT
    VI_DataPtr : POINTER TO BYTE;
    VI_Size : UDINT;
  END_VAR
  VAR
    L_k : UDINT;
    L_CRC : DWORD := 16#FFFFFFFF;
  END_VAR
                  InitTable();

IF VI_DataPtr = 0 OR VI_Size = 0 THEN
    Calculate := 0;
    RETURN;
END_IF;

FOR L_k := 0 TO VI_Size - 1 DO
    L_CRC := L_Table[TO_INT((L_CRC XOR VI_DataPtr[TO_INT(L_k)]) AND 16#FF)] XOR SHR(L_CRC, 8);
END_FOR;

Calculate := L_CRC XOR 16#FFFFFFFF;
                
END_METHOD
END_FUNCTION_BLOCK

FUNCTION_BLOCK FB_Debug_Logger
  VAR_INPUT
    VI_Config : ST_Debug_Logger_Config;
    VI_System_Time_MS : UDINT;
    VI_Floor_Temps : ARRAY[1..16] OF REAL;
    VI_Pump_Currents : ARRAY[1..5] OF REAL;
    VI_Error_Code : UDINT;
  END_VAR
  VAR
    L_buffer : ARRAY[1..1000] OF ST_Debug_Log_Record;
    L_write_idx : INT := 1;
    L_last_log_time : UDINT;
    L_i : INT;
  END_VAR

            // Цикл логирования
IF VI_Config.enabled AND (VI_System_Time_MS - L_last_log_time >= VI_Config.sampling_period_ms) THEN
    L_last_log_time := VI_System_Time_MS;
    
    // Логируем температуры (если изменились или по таймауту)
    FOR L_i := 1 TO 16 DO
        L_buffer[L_write_idx].timestamp_ms := VI_System_Time_MS;
        L_buffer[L_write_idx].level := E_Debug_Log_Level.LOG_LEVEL_VERBOSE;
        L_buffer[L_write_idx].source_id := TO_BYTE(L_i);
        L_buffer[L_write_idx].value_real := VI_Floor_Temps[L_i];
        L_buffer[L_write_idx].text := 'Floor Temp Update';
        
        L_write_idx := (L_write_idx MOD 1000) + 1;
    END_FOR;

    // Логируем ошибки
    IF VI_Error_Code <> 0 THEN
        L_buffer[L_write_idx].timestamp_ms := VI_System_Time_MS;
        L_buffer[L_write_idx].level := E_Debug_Log_Level.LOG_LEVEL_MINIMAL;
        L_buffer[L_write_idx].event_code := TO_WORD(VI_Error_Code);
        L_buffer[L_write_idx].text := 'System Error Detected';
        L_write_idx := (L_write_idx MOD 1000) + 1;
    END_IF;
END_IF;

          
END_FUNCTION_BLOCK

FUNCTION_BLOCK FB_Device_Predictive_Diag
  VAR_INPUT
    VI_Current_Value : REAL;  (* Текущий ток или время *)
    VI_Nominal_Value : REAL;  (* Эталонное значение *)
    VI_Is_Running : BOOL;
    VI_Reset_Stats : BOOL;
  END_VAR
  VAR_IN_OUT
    VIO_Health_Data : ST_Device_Health;
  END_VAR
  VAR
    L_Prev_Running : BOOL;
    L_Current_Sum : REAL;
    L_Sample_Count : UDINT;
  END_VAR

            // 1. Счётчик пусков и замер пускового тока
IF VI_Is_Running AND NOT L_Prev_Running THEN
    VIO_Health_Data.Starts_Count := VIO_Health_Data.Starts_Count + 1;
    VIO_Health_Data.Last_Start_Current := VI_Current_Value;
    
    // Обновление среднего пускового тока
    L_Sample_Count := L_Sample_Count + 1;
    L_Current_Sum := L_Current_Sum + VI_Current_Value;
    VIO_Health_Data.Avg_Start_Current := L_Current_Sum / UDINT_TO_REAL(L_Sample_Count);
END_IF;

// 2. Анализ отклонения (п. 12.1 ТЗ)
IF VI_Is_Running THEN
    // Если ток выше номинала на 50% - снижаем здоровье
    IF VI_Current_Value > (VI_Nominal_Value * 1.5) THEN
        IF VIO_Health_Data.Health_Score > 0 THEN
            VIO_Health_Data.Health_Score := VIO_Health_Data.Health_Score - 1;
        END_IF;
    END_IF;
END_IF;

// 3. Генерация предупреждения
IF VIO_Health_Data.Health_Score < 20 THEN
    VIO_Health_Data.Maintenance_Required := TRUE;
    VIO_Health_Data.Warning_Message := 'Критический износ: проверьте механику';
ELSIF VIO_Health_Data.Health_Score < 60 THEN
    VIO_Health_Data.Warning_Message := 'Предупреждение: повышенное трение';
END_IF;

L_Prev_Running := VI_Is_Running;

          
END_FUNCTION_BLOCK

FUNCTION_BLOCK FB_DHW_Manager
  VAR_INPUT
    VI_System_Time_MS : UDINT;
    VI_IsActivePLC : BOOL;
    VI_Temp : REAL;
    VI_Pressure : REAL;
    VI_Config : ST_DHW_Config;
    VI_Maintenance : ST_Component_Maintenance;
  END_VAR
  VAR_OUTPUT
    VO_Status : ST_DHW_Status;
    VO_Heating_Pump : BOOL;
    VO_Circ_Pump : BOOL;
  END_VAR
  VAR
    L_Current_TOD : TOD;
    L_Legionella_Active : BOOL;
    L_Last_Good_Temp : REAL := 55;
  END_VAR

            IF NOT VI_IsActivePLC THEN RETURN; END_IF;

L_DHW_V2_Shadow_Diff_Found := FALSE;
L_DHW_V2_Switch_Enabled := TRUE;
L_DHW_V2_Path_Ready := FALSE;
L_DHW_Using_Legacy_Fallback := TRUE;

GVL_STATE.G_DHW_IO_Fault := FALSE;
GVL_STATE.G_DHW_Sensor_Fault := FALSE;
GVL_STATE.G_DHW_Subsystem_Degraded := FALSE;

IF VI_Emergency_Stop THEN
    VO_Heating_Pump := FALSE;
    VO_Circ_Pump := FALSE;
    VO_Status.Warning := FALSE;
    VO_Status.Error := TRUE;
    VO_Status.Error_ID := GVL_CONFIG.ERR_DHW_IO_OFFLINE; // временно используем общий аварийный код до детализации safety-кодов
    VO_Status.Heating_Pump_On := FALSE;
    VO_Status.Circ_Pump_On := FALSE;
    RETURN;
END_IF;

// Фиксация текущего времени
L_Current_TOD := VI_Current_TOD;

// ========================================
// DHW POLICY LAYER
// ========================================
L_Policy_Safe_Stop := (VI_System_Mode = E_System_Operating_Mode.MODE_SAFE_STOP);
L_Policy_Freeze_Protection := (VI_System_Mode = E_System_Operating_Mode.MODE_FREEZE_PROTECTION);
L_Policy_Degraded := (VI_System_Mode = E_System_Operating_Mode.MODE_DEGRADED);
L_Target_Temp_Adjusted := VI_Config.Target_Temp;
IF L_Policy_Degraded THEN
    L_Target_Temp_Adjusted := VI_Config.Target_Temp - VI_Config.Degraded_Target_Delta;
END_IF;

// ========================================
// DHW POLICY OVERRIDE
// ========================================
IF L_Policy_Safe_Stop THEN
    VO_Heating_Pump := FALSE;
    VO_Circ_Pump := FALSE;
    RETURN;
END_IF;

IF L_Policy_Freeze_Protection THEN
    VO_Heating_Pump := FALSE;
    VO_Circ_Pump := FALSE;
    RETURN;
END_IF;

// Сброс признака выполнения термодезинфекции при смене дня.
IF L_Last_Legionella_Day <> VI_Current_Day_Of_Week THEN
    L_Legionella_Done_Today := FALSE;
    L_Last_Legionella_Day := VI_Current_Day_Of_Week;
END_IF;

// Базовый сброс незащёлкнутых статусных флагов на текущий цикл.
// Критические ошибки ниже могут зафиксироваться и завершить выполнение через RETURN.
VO_Status.Warning := FALSE;
VO_Status.Error := FALSE;
VO_Status.Error_ID := 0;

// Сброс ошибок
IF VI_Reset_Errors THEN
    L_Error_Latched := FALSE;
    L_Error_ID_Latched := 0;
END_IF;

// Проверка связи с модулями ввода-вывода
FOR L_i := 1 TO GVL_CONSTANTS.C_MAX_MODULES DO
    IF NOT VI_IO_Modules_Online[L_i] THEN
        L_Error_Latched := TRUE;
        GVL_STATE.G_DHW_IO_Fault := TRUE;
        L_Error_ID_Latched := GVL_CONFIG.ERR_DHW_IO_OFFLINE; // Потеря связи с модулями ввода-вывода
    END_IF;
END_FOR;

// 1. Обработка неисправностей датчиков и сервисных режимов (ТЗ 7.0)
fbTempValidator(
    VI_Value := VI_Temp,
    VI_Min_Valid := 0.0,
    VI_Max_Valid := 100.0,
    VI_Fallback_Mode := 0,
    VI_Default_Value := 55.0
);

fbPressValidator(
    VI_Value := VI_Pressure,
    VI_Min_Valid := 0.0,
    VI_Max_Valid := 10.0,
    VI_Fallback_Mode := 0
);

VO_Status.Temp := fbTempValidator.VO_Value;
VO_Status.Pressure := fbPressValidator.VO_Value;

// Сохраняем последнее достоверное значение температуры ГВС.
// Используется только для диагностики/сервиса, не для fallback-управления.
IF NOT fbTempValidator.VO_Error THEN
    L_Last_Good_Temp := VO_Status.Temp;
END_IF;

IF fbTempValidator.VO_Error THEN
    GVL_STATE.G_DHW_Sensor_Fault := TRUE;
    L_Error_Latched := TRUE;
    L_Error_ID_Latched := GVL_CONFIG.ERR_DHW_TEMP_SENSOR_FAULT; // Критическая ошибка датчика температуры
ELSIF (VO_Status.Pressure < 1.0 OR VO_Status.Pressure > 4.0) AND NOT fbPressValidator.VO_Error THEN
    L_Error_Latched := TRUE;
    L_Error_ID_Latched := GVL_CONFIG.ERR_DHW_PRESSURE_OUT_OF_RANGE; // Давление вне нормы
END_IF;

IF L_Error_Latched THEN
    // Критическая ошибка: переход в безопасное состояние с полной остановкой насосов.
    VO_Heating_Pump := FALSE;
    VO_Circ_Pump := FALSE;
    VO_Status.Warning := FALSE;
    VO_Status.Error := TRUE;
    VO_Status.Error_ID := L_Error_ID_Latched;
    VO_Status.Heating_Pump_On := FALSE;
    VO_Status.Circ_Pump_On := FALSE;
    RETURN;
END_IF;

// Ошибка датчика давления не останавливает ГВС,
// но переводит подсистему в режим предупреждения (degraded mode).
IF fbPressValidator.VO_Error THEN
    GVL_STATE.G_DHW_Sensor_Fault := TRUE;
    GVL_STATE.G_DHW_Subsystem_Degraded := TRUE;
    VO_Status.Warning := TRUE;
    VO_Status.Error := FALSE;
    VO_Status.Error_ID := GVL_CONFIG.ERR_DHW_PRESSURE_SENSOR_FAULT;
END_IF;

// 2. Логика поддержания температуры воды в бойлере (Нагрев)
// На этом этапе FB уже выполняется только на активном ПЛК.
    
// Термическая дезинфекция (Легионелла)
IF VI_Config.Anti_Legionella_Enabled
   AND (VI_Current_Day_Of_Week = VI_Config.Anti_Legionella_Day)
   AND (L_Current_TOD >= TOD#02:00)
   AND (L_Current_TOD <= TOD#04:00)
   AND NOT L_Legionella_Done_Today THEN
    L_Legionella_Active := TRUE;
ELSE
    L_Legionella_Active := FALSE;
END_IF;

L_Legionella_Timer(IN := L_Legionella_Active AND VO_Status.Temp >= 70.0, PT := T#30m, VI_System_Time_MS := VI_System_Time_MS);
IF L_Legionella_Timer.Q THEN
    L_Legionella_Active := FALSE; // Дезинфекция завершена
    L_Legionella_Done_Today := TRUE; // Повторно в те же сутки не запускать
END_IF;

// Двухпозиционное регулирование с гистерезисом
IF L_Legionella_Active THEN
    IF VO_Status.Temp < 70.0 THEN
        VO_Heating_Pump := TRUE;
    ELSIF VO_Status.Temp > 72.0 THEN
        VO_Heating_Pump := FALSE;
    END_IF;
ELSE
    IF VO_Status.Temp < (L_Target_Temp_Adjusted - VI_Config.Hysteresis) THEN
        VO_Heating_Pump := TRUE;
    ELSIF VO_Status.Temp > (L_Target_Temp_Adjusted + VI_Config.Hysteresis) THEN
        VO_Heating_Pump := FALSE;
    END_IF;
END_IF;

// 3. Управление циркуляционным насосом ГВС по расписанию
// Рециркуляция обеспечивает мгновенное наличие горячей воды у потребителя
VO_Circ_Pump := VI_Config.Circulation_Schedule_Enabled AND NOT (VI_Config.Night_Mode_Enabled AND (L_Current_TOD < VI_Config.Circulation_Start OR L_Current_TOD > VI_Config.Circulation_End));

// Формирование статусных данных для визуализации.
// К этому моменту статус уже консистентен:
// - Error = критическая ошибка с остановкой ГВС
// - Warning = деградация без остановки
VO_Status.Heating_Pump_On := VO_Heating_Pump;
VO_Status.Circ_Pump_On := VO_Circ_Pump;

// ========================================
// DHW V2 shadow execution (phase2)
// ========================================
fbDHWV2Staging(
    VI_Tank_ID := 1,
    VI_Enable := TRUE,
    VI_Target_Temp := VI_Config.Target_Temp,
    VI_Pump_Enable := VO_Heating_Pump,
    VI_Heating_Priority := FALSE,

    VI_Is_Active := TRUE,
    VI_Tank_Temp := VO_Status.Temp,
    VI_Supply_Temp := VO_Status.Temp,
    VI_Return_Temp := VO_Status.Temp,
    VI_Pump_Actual := VO_Heating_Pump,
    VI_Alarm_Active := VO_Status.Error,

    VO_Command_Shadow => L_DHW_V2_Command_Shadow,
    VO_State_Shadow => L_DHW_V2_State_Shadow
);

// ========================================
// DHW V2 shadow validation
// ========================================
IF ABS(VO_Heating_Pump - L_DHW_V2_Command_Shadow.Pump_Enable) > 0.1 THEN
    L_DHW_V2_Shadow_Diff_Found := TRUE;
END_IF;
IF ABS(VO_Status.Temp - L_DHW_V2_State_Shadow.Tank_Temp) > 0.1 THEN
    L_DHW_V2_Shadow_Diff_Found := TRUE;
END_IF;
IF ABS(VO_Status.Pressure - L_DHW_V2_State_Shadow.Supply_Temp) > 0.1 THEN
    L_DHW_V2_Shadow_Diff_Found := TRUE;
END_IF;

// Guarded DHW V2 enable
IF L_DHW_V2_Switch_Enabled THEN
    IF NOT L_DHW_V2_Shadow_Diff_Found THEN
        L_DHW_V2_Path_Ready := TRUE;
        L_DHW_Using_Legacy_Fallback := FALSE;
    ELSE
        L_DHW_V2_Path_Ready := FALSE;
        L_DHW_Using_Legacy_Fallback := TRUE;
    END_IF;
ELSE
    L_DHW_V2_Path_Ready := FALSE;
    L_DHW_Using_Legacy_Fallback := TRUE;
END_IF;

END_FUNCTION_BLOCK
// >>> BULK_SYNC_ANCHOR: FB_DHW_Manager <<<

          
END_FUNCTION_BLOCK

FUNCTION_BLOCK FB_Emergency_Valve_Open
  VAR_INPUT
    VI_Fire_Alarm : BOOL;
    VI_Gas_Alarm : BOOL;
  END_VAR
  VAR_OUTPUT
    VO_Open_Cmd : BOOL;
  END_VAR

            // Приоритетное открытие при любой серьезной аварии
VO_Open_Cmd := VI_Fire_Alarm OR VI_Gas_Alarm;

          
END_FUNCTION_BLOCK

FUNCTION_BLOCK FB_Exhaust_Ventilation_Controller
  VAR_INPUT
    VI_Humidity : REAL;
    VI_CO2 : REAL;
    VI_Config : ST_Ventilation_Unit_Config;
  END_VAR
  VAR_OUTPUT
    VO_Fan_Speed : BYTE;
  END_VAR

            IF VI_Humidity > VI_Config.Threshold_Hum THEN
    VO_Fan_Speed := 100;
ELSIF VI_CO2 > 800.0 THEN
    VO_Fan_Speed := 70;
ELSE
    VO_Fan_Speed := 40;
END_IF;

          
END_FUNCTION_BLOCK

FUNCTION_BLOCK FB_Flood_Detector
  VAR_INPUT
    VI_Sensors : ARRAY[1..12] OF BOOL;
    VI_IsActivePLC : BOOL;
  END_VAR
  VAR_OUTPUT
    VO_Flood_Alarm : BOOL;
    VO_Close_Valve_35 : BOOL;
    VO_Close_Valve_36 : BOOL;
  END_VAR
  VAR
    L_i : INT;
  END_VAR

            VO_Flood_Alarm := FALSE;
VO_Close_Valve_35 := FALSE;
VO_Close_Valve_36 := FALSE;

FOR L_i := 1 TO 12 DO
    IF VI_Sensors[L_i] THEN
        VO_Flood_Alarm := TRUE;
        IF VI_IsActivePLC THEN
            // Логика п. 4.2: Зона 2 (4-5) и Зона 3 (6-7) делят клапан 36
            IF L_i >= 4 AND L_i <= 7 THEN
                VO_Close_Valve_36 := TRUE;
            ELSIF L_i >= 1 AND L_i <= 3 THEN
                VO_Close_Valve_35 := TRUE;
            END_IF;
        END_IF;
    END_IF;
END_FOR;

          
END_FUNCTION_BLOCK

FUNCTION_BLOCK FB_FloorHeating_Controller
  VAR_INPUT
    VI_Current_Temp : REAL;
    VI_Config : ST_FloorHeating_Circuit_Config;
    VI_Tariff : ST_Tariff_Config;
    VI_Current_Hour : UINT;
    VI_IsActivePLC : BOOL;
  END_VAR
  VAR_OUTPUT
    VO_Pump_Run : BOOL;
    VO_Valve_Pos : REAL;  (* 0..10V *)
    VO_Effective_Setpoint : REAL;
  END_VAR
  VAR
    L_Is_Night : BOOL;
  END_VAR

            // 1. Определение активного тарифа
IF VI_Tariff.Enabled THEN
    IF VI_Tariff.Night_Start_Hour > VI_Tariff.Night_End_Hour THEN
        // Переход через полночь (например, 23:00 - 07:00)
        L_Is_Night := (VI_Current_Hour >= VI_Tariff.Night_Start_Hour) OR (VI_Current_Hour < VI_Tariff.Night_End_Hour);
    ELSE
        // В пределах одного дня
        L_Is_Night := (VI_Current_Hour >= VI_Tariff.Night_Start_Hour) AND (VI_Current_Hour < VI_Tariff.Night_End_Hour);
    END_IF;
ELSE
    L_Is_Night := FALSE;
END_IF;

// 2. Расчет эффективной уставки
VO_Effective_Setpoint := VI_Config.design_temp;
IF L_Is_Night THEN
    VO_Effective_Setpoint := VO_Effective_Setpoint + VI_Tariff.Boost_Delta;
END_IF;

// 3. Простая логика управления (гистерезис)
IF VI_IsActivePLC THEN
    IF VI_Current_Temp < (VO_Effective_Setpoint - 0.5) THEN
        VO_Pump_Run := TRUE;
        VO_Valve_Pos := 10.0;
    ELSIF VI_Current_Temp > (VO_Effective_Setpoint + 0.5) THEN
        VO_Pump_Run := FALSE;
        VO_Valve_Pos := 0.0;
    END_IF;
END_IF;

          
END_FUNCTION_BLOCK

FUNCTION_BLOCK FB_FloorHeating_Freeze_Protection
  VAR_INPUT
    VI_Floor_Temps : ARRAY[1..16] OF REAL;
    VI_Outdoor_Temp : REAL;
    VI_Threshold : REAL := 7;
  END_VAR
  VAR_OUTPUT
    VO_Freeze_Alert : BOOL;
    VO_Pump_Force_On : BOOL;
  END_VAR
  VAR
    L_i : INT;
  END_VAR

            VO_Freeze_Alert := FALSE;
VO_Pump_Force_On := FALSE;

FOR L_i := 1 TO 16 DO
    IF VI_Floor_Temps[L_i] < VI_Threshold THEN
        VO_Freeze_Alert := TRUE;
        VO_Pump_Force_On := TRUE;
        RETURN;
    END_IF;
END_FOR;

IF VI_Outdoor_Temp < -5.0 THEN
    VO_Pump_Force_On := TRUE;
END_IF;

          
END_FUNCTION_BLOCK

FUNCTION_BLOCK FB_FloorHeating_Overheat_Protection
  VAR_INPUT
    VI_Temps : ARRAY[1..16] OF REAL;
    VI_Threshold : REAL := 45;
  END_VAR
  VAR_OUTPUT
    VO_Overheat_Detected : BOOL;
    VO_Locked_Circuits : ARRAY[1..16] OF BOOL;
  END_VAR
  VAR
    L_i : INT;
  END_VAR

            VO_Overheat_Detected := FALSE;
FOR L_i := 1 TO 16 DO
    IF VI_Temps[L_i] > VI_Threshold THEN
        VO_Overheat_Detected := TRUE;
        VO_Locked_Circuits[L_i] := TRUE;
    END_IF;
END_FOR;

          
END_FUNCTION_BLOCK

FUNCTION_BLOCK FB_Gas_Methane_Detector
  VAR_INPUT
    VI_Methane_LEL : REAL;
    VI_Threshold_Alarm : REAL := 20;
  END_VAR
  VAR_OUTPUT
    VO_Alarm_Active : BOOL;
    VO_Close_Valve : BOOL;
  END_VAR

            VO_Alarm_Active := (VI_Methane_LEL >= VI_Threshold_Alarm);
VO_Close_Valve := VO_Alarm_Active;

          
END_FUNCTION_BLOCK

FUNCTION_BLOCK FB_Gas_Smoke_Manager
  VAR_INPUT
    VI_System_Time_MS : UDINT;
    VI_IsActivePLC : BOOL;
    VI_Methane_LEL : ARRAY[1..2] OF REAL;
    VI_CO_PPM : ARRAY[1..8] OF REAL;
    VI_Smoke_Sensors : ARRAY[1..6] OF BOOL;
    VI_Mute_Request : BOOL;
  END_VAR
  VAR_OUTPUT
    VO_Gas_Alarm : BOOL;
    VO_Fire_Alarm : BOOL;
    VO_Siren_Active : BOOL;
    VO_Gas_Valve_Close : BOOL;
    VO_Boiler_Stop : BOOL;
    VO_Vent_PV3_Boost : BOOL;  (* ТЗ 5.1 (ПВ-3 при 10% LEL) *)
    VO_Supply_100_Req : BOOL;  (* ТЗ 6.4 (Метан >20%) *)
    VO_Exhaust_100_Req : BOOL;  (* ТЗ 6.4 (Пожар) *)
    VO_Supply_80_Req : BOOL;  (* ТЗ 5.4 (CO) *)
    VO_Status_Msg : STRING(200);
  END_VAR
  VAR
    L_Methane_Max : REAL;
    L_CO_Max : REAL;
    L_Smoke_Active : BOOL;
    L_Smoke_Timer : ARRAY[1..6] OF TON;
    L_Mute_Timer : TON;
    L_Muted : BOOL;
    L_Mute_Count : UINT;  (* ТЗ 5.5 *)
    L_i : INT;
    L_j : INT;
    L_Smoke_Count : UINT;
    L_CO_Timer_30ppm : TON;  (* 8 часов *)
    L_CO_Timer_70ppm : TON;  (* 1 час *)
    L_CO_Timer_400ppm : TON;  (* 15 минут *)
  END_VAR

            IF NOT VI_IsActivePLC THEN RETURN; END_IF;

// Reset outputs
VO_Smoke_Detected := FALSE;
VO_Gas_Detected := FALSE;
VO_CO_Warning_Level := FALSE;
VO_CO_Alarm_Level := FALSE;

VO_Siren_Active := FALSE;
VO_Gas_Valve_Close := FALSE;
VO_Boiler_Stop := FALSE;
VO_Vent_PV3_Boost := FALSE;
VO_Supply_100_Req := FALSE;
VO_Exhaust_100_Req := FALSE;
VO_Supply_80_Req := FALSE;
VO_Vent_Stop := FALSE;
VO_Status_Msg := 'ОК';

// --- Methane ---
L_Methane_Max := 0.0;
FOR L_i := 1 TO GVL_CONSTANTS.C_MAX_METHANE_SENSORS DO
    IF VI_Methane_LEL[L_i] > L_Methane_Max THEN
        L_Methane_Max := VI_Methane_LEL[L_i];
    END_IF;
END_FOR;

IF L_Methane_Max >= 10.0 THEN
    VO_Vent_PV3_Boost := TRUE;
END_IF;

IF L_Methane_Max >= 20.0 THEN
    VO_Gas_Detected := TRUE;
    VO_Gas_Valve_Close := TRUE;
    VO_Boiler_Stop := TRUE;
    VO_Supply_100_Req := TRUE;
END_IF;

// --- CO ---
L_CO_Max := 0.0;
FOR L_i := 1 TO GVL_CONSTANTS.C_MAX_CO_SENSORS DO
    IF VI_CO_PPM[L_i] > L_CO_Max THEN
        L_CO_Max := VI_CO_PPM[L_i];
    END_IF;
END_FOR;

L_CO_Level_30 := (L_CO_Max >= 30.0);
L_CO_Level_70 := (L_CO_Max >= 70.0);
L_CO_Level_400 := (L_CO_Max >= 400.0);

L_CO_Timer_30ppm(IN := L_CO_Level_30, PT := T#8h, VI_System_Time_MS := VI_System_Time_MS);
L_CO_Timer_70ppm(IN := L_CO_Level_70, PT := T#1h, VI_System_Time_MS := VI_System_Time_MS);
L_CO_Timer_400ppm(IN := L_CO_Level_400, PT := T#15m, VI_System_Time_MS := VI_System_Time_MS);

IF L_CO_Timer_30ppm.Q THEN
    VO_CO_Warning_Level := TRUE;
    VO_Supply_80_Req := TRUE;
END_IF;

IF L_CO_Timer_70ppm.Q OR L_CO_Timer_400ppm.Q THEN
    VO_CO_Alarm_Level := TRUE;
    VO_Supply_80_Req := TRUE;
END_IF;

// --- Smoke ---
L_Smoke_Count := 0;
L_Smoke_Active := FALSE;

FOR L_i := 1 TO GVL_CONSTANTS.C_MAX_SMOKE_SENSORS DO
    L_Smoke_Timer[L_i](IN := VI_Smoke_Sensors[L_i], PT := T#30s, VI_System_Time_MS := VI_System_Time_MS);

    IF VI_Smoke_Sensors[L_i] THEN
        L_Smoke_Count := L_Smoke_Count + 1;
    END_IF;

    IF L_Smoke_Timer[L_i].Q OR (L_Smoke_Count >= 2) THEN
        L_Smoke_Active := TRUE;
    END_IF;
END_FOR;

IF L_Smoke_Active THEN
    VO_Smoke_Detected := TRUE;
    VO_Vent_Stop := TRUE;
    VO_Boiler_Stop := TRUE;
END_IF;

// Status
IF VO_Smoke_Detected THEN
    VO_Status_Msg := 'ПОЖАР';
ELSIF VO_Gas_Detected THEN
    VO_Status_Msg := 'УТЕЧКА ГАЗА';
ELSIF VO_CO_Alarm_Level THEN
    VO_Status_Msg := 'КРИТИЧЕСКИЙ CO';
ELSIF VO_CO_Warning_Level THEN
    VO_Status_Msg := 'ПОВЫШЕННЫЙ CO';
ELSE
    VO_Status_Msg := 'ОК';
END_IF;
// >>> BULK_SYNC_ANCHOR: FB_Gas_Smoke_Manager <<<

          
END_FUNCTION_BLOCK

FUNCTION_BLOCK FB_Gas_Valve_Controller IMPLEMENTS IValveController
  VAR_INPUT
    VI_System_Time : UDINT;
    VI_IsActivePLC : BOOL;
    VI_Gas_Alarm : BOOL;
    VI_Config : ST_Gas_Valve_Configuration;
  END_VAR
  VAR_OUTPUT
    VO_Valve_Closed : BOOL;
    VO_Status_Msg : STRING(200);
  END_VAR

            // При аварии газа - немедленное закрытие
IF VI_Gas_Alarm AND VI_IsActivePLC THEN
    VO_Valve_Closed := TRUE;
    VO_Status_Msg := 'ГАЗОВЫЙ КЛАПАН ЗАКРЫТ ПО АВАРИИ';
END_IF;
          

METHOD CloseValve : BOOL
  VAR_INPUT
    VI_Operator_ID : STRING(10);
    VI_Force : BOOL;
  END_VAR
                  VO_Valve_Closed := TRUE;
CloseValve := TRUE;
                
END_METHOD

METHOD GetStatus : BYTE
                  GetStatus := TO_BYTE(SEL(VO_Valve_Closed, 0, 1));
                
END_METHOD

METHOD OpenValve : BOOL
  VAR_INPUT
    VI_Operator_ID : STRING(10);
    VI_Force : BOOL;
  END_VAR
                  IF VI_IsActivePLC OR VI_Force THEN
    VO_Valve_Closed := FALSE;
    OpenValve := TRUE;
END_IF;
                
END_METHOD
END_FUNCTION_BLOCK

FUNCTION_BLOCK FB_Gateway_Interface
  VAR_INPUT
    VI_System_Time_MS : UDINT;
    VI_Local_PLC_Role : E_PLC_ROLE;
    VI_Incoming_Command : ST_Gateway_Command;
    VI_Command_Received : BOOL;
    VI_FloorHeating_Temps : ARRAY[1..16] OF REAL;  (* Состояния системы *)
    VI_Room_Temps : ARRAY[1..16] OF REAL;
    VI_Zone_Valve_States : ARRAY[1..16] OF BOOL;
    VI_Manifold_Pressures : ARRAY[1..5] OF REAL;
    VI_Manifold_Pump_States : ARRAY[1..5] OF BOOL;
    VI_Outdoor_Temp : REAL;
    VI_Security_Armed : BOOL;
    VI_Flood_Alarm_Active : BOOL;
    VI_Gas_Alarm_Active : BOOL;
    VI_Fire_Alarm_Active : BOOL;
    VI_Methane_Concentration : REAL;
    VI_Lighting_Base_Levels : ARRAY[1..16] OF BYTE;
    VI_Socket_States : ARRAY[1..36] OF BOOL;
    VI_Blinds_Positions : ARRAY[1..20] OF BYTE;
    VI_Active_Scenario : E_SCENARIO_TYPE;
  END_VAR
  VAR_OUTPUT
    VO_Modbus_Registers : ARRAY[0..200] OF WORD;  (* Расширенный диапазон *)
    VO_Lighting_Override : ARRAY[1..16] OF BYTE;
    VO_Socket_Override : ARRAY[1..36] OF BOOL;
    VO_Data_Ready : BOOL;
    VO_HMI_Status_Message : STRING(200);
  END_VAR
  VAR
    L_last_update_time : UDINT;
    L_i : INT;
    L_j : INT;
    L_idx : INT;
    L_tmp_word : WORD;
  END_VAR

            // Отправка уведомлений в Telegram (ТЗ 10.2)
VO_Send_Telegram := FALSE;
IF VI_Fire_Alarm_Active AND NOT L_Prev_Fire THEN
    VO_Telegram_Msg := 'ВНИМАНИЕ! ПОЖАРНАЯ ТРЕВОГА!';
    VO_Send_Telegram := TRUE;
END_IF;
IF VI_Gas_Alarm_Active AND NOT L_Prev_Gas THEN
    VO_Telegram_Msg := 'ВНИМАНИЕ! УТЕЧКА ГАЗА!';
    VO_Send_Telegram := TRUE;
END_IF;
IF VI_Flood_Alarm_Active AND NOT L_Prev_Flood THEN
    VO_Telegram_Msg := 'ВНИМАНИЕ! ПРОТЕЧКА ВОДЫ!';
    VO_Send_Telegram := TRUE;
END_IF;
IF VI_Security_Armed AND NOT L_Prev_Security THEN
    VO_Telegram_Msg := 'ОХРАНА ВКЛЮЧЕНА';
    VO_Send_Telegram := TRUE;
ELSIF NOT VI_Security_Armed AND L_Prev_Security THEN
    VO_Telegram_Msg := 'ОХРАНА ОТКЛЮЧЕНА';
    VO_Send_Telegram := TRUE;
END_IF;

L_Prev_Fire := VI_Fire_Alarm_Active;
L_Prev_Gas := VI_Gas_Alarm_Active;
L_Prev_Flood := VI_Flood_Alarm_Active;
L_Prev_Security := VI_Security_Armed;

// Обновление данных Modbus (раз в 1 сек)
IF F_TimeDiff(VI_System_Time_MS, L_last_update_time) >= GVL_CONSTANTS.C_MS_IN_SECOND THEN
    L_last_update_time := VI_System_Time_MS;
    
    // 0: Статус ПЛК и Аварии
    L_tmp_word := 0;
    IF VI_Local_PLC_Role = E_PLC_ROLE.ROLE_ACTIVE THEN L_tmp_word := L_tmp_word OR 1; END_IF;
    IF VI_Security_Armed THEN L_tmp_word := L_tmp_word OR 2; END_IF;
    IF VI_Flood_Alarm_Active THEN L_tmp_word := L_tmp_word OR 4; END_IF;
    IF VI_Gas_Alarm_Active THEN L_tmp_word := L_tmp_word OR 8; END_IF;
    IF VI_Fire_Alarm_Active THEN L_tmp_word := L_tmp_word OR 16; END_IF;
    VO_Modbus_Registers[0] := L_tmp_word;

    // 1-16: Температуры пола (x10)
    FOR L_i := 1 TO GVL_CONSTANTS.C_MAX_HEATING_CIRCUITS DO
        VO_Modbus_Registers[L_i] := TO_WORD(TO_INT(VI_FloorHeating_Temps[L_i] * 10.0));
    END_FOR;

    // 17-32: Температуры помещений (x10)
    FOR L_i := 1 TO GVL_CONSTANTS.C_MAX_CLIMATE_ZONES DO
        VO_Modbus_Registers[16 + L_i] := TO_WORD(TO_INT(VI_Room_Temps[L_i] * 10.0));
    END_FOR;

    // 33: Состояние клапанов зон (битовая маска 1-16)
    L_tmp_word := 0;
    FOR L_i := 1 TO GVL_CONSTANTS.C_MAX_HEATING_CIRCUITS DO
        IF VI_Zone_Valve_States[L_i] THEN
            L_tmp_word := L_tmp_word OR SHL(TO_WORD(1), L_i - 1);
        END_IF;
    END_FOR;
    VO_Modbus_Registers[33] := L_tmp_word;

    // 34-38: Давление в коллекторах (x100)
    FOR L_i := 1 TO GVL_CONSTANTS.C_MAX_MANIFOLDS DO
        VO_Modbus_Registers[33 + L_i] := TO_WORD(TO_INT(VI_Manifold_Pressures[L_i] * 100.0));
    END_FOR;

    // 40-55: Базовое освещение
    FOR L_i := 1 TO GVL_CONSTANTS.C_MAX_LIGHTING_ZONES DO
        VO_Modbus_Registers[39 + L_i] := TO_WORD(VI_Lighting_Base_Levels[L_i]);
    END_FOR;

    // 60-79: Положение штор (20 шт)
    FOR L_i := 1 TO GVL_CONSTANTS.C_MAX_BLINDS DO
        VO_Modbus_Registers[59 + L_i] := TO_WORD(VI_Blinds_Positions[L_i]);
    END_FOR;

    // 80-82: Розетки (битовая маска, 36 розеток -> 3 WORD)
    FOR L_i := 0 TO (GVL_CONSTANTS.C_MAX_SOCKETS - 1) / 16 DO
        L_tmp_word := 0;
        FOR L_j := 1 TO 16 DO
            L_idx := (L_i * 16) + L_j;
            IF L_idx <= GVL_CONSTANTS.C_MAX_SOCKETS THEN
                IF VI_Socket_States[L_idx] THEN
                    L_tmp_word := L_tmp_word OR SHL(TO_WORD(1), L_j - 1);
                END_IF;
            END_IF;
        END_FOR;
        VO_Modbus_Registers[79 + L_i] := L_tmp_word;
    END_FOR;

    // 100-102: 2FA Request and Code
    VO_Modbus_Registers[100] := SEL(VI_Send_2FA_Req, 0, 1);
    IF VI_Send_2FA_Req THEN
        L_Code_UDINT := STRING_TO_UDINT(VI_2FA_Code);
        VO_Modbus_Registers[101] := TO_WORD(L_Code_UDINT AND 16#FFFF);
        VO_Modbus_Registers[102] := TO_WORD(SHR(L_Code_UDINT, 16));
    ELSE
        VO_Modbus_Registers[101] := 0;
        VO_Modbus_Registers[102] := 0;
    END_IF;

    VO_Data_Ready := TRUE;
END_IF;

// Обработка входящих команд
VO_Arm_Req := FALSE;
VO_Disarm_Req := FALSE;
VO_Set_Scenario_Req := FALSE;
VO_Set_Temp_Req := FALSE;
VO_Set_Vent_Req := FALSE;
VO_Reset_Errors_Req := FALSE;
VO_Set_Config_Req := FALSE;
VO_Sync_Time_Req := FALSE;
L_Has_Command_To_Process := FALSE;

// 1. Прием команды и буферизация
IF VI_Command_Received THEN
    IF VI_Local_PLC_Role = E_PLC_ROLE.ROLE_ACTIVE THEN
        // Если активен, обрабатываем сразу
        L_Process_Command := VI_Incoming_Command;
        L_Has_Command_To_Process := TRUE;
    ELSE
        // Если резервный, добавляем в буфер
        IF L_Buffer_Count < GVL_CONSTANTS.C_MAX_GATEWAY_COMMANDS THEN
            L_Command_Buffer[L_Buffer_Head] := VI_Incoming_Command;
            L_Buffer_Head := L_Buffer_Head + 1;
            IF L_Buffer_Head > GVL_CONSTANTS.C_MAX_GATEWAY_COMMANDS THEN L_Buffer_Head := 1; END_IF;
            L_Buffer_Count := L_Buffer_Count + 1;
        END_IF;
    END_IF;
END_IF;

// 2. Извлечение из буфера при переходе в активный режим
IF NOT L_Has_Command_To_Process AND (VI_Local_PLC_Role = E_PLC_ROLE.ROLE_ACTIVE) AND (L_Buffer_Count > 0) THEN
    L_Process_Command := L_Command_Buffer[L_Buffer_Tail];
    L_Buffer_Tail := L_Buffer_Tail + 1;
    IF L_Buffer_Tail > GVL_CONSTANTS.C_MAX_GATEWAY_COMMANDS THEN L_Buffer_Tail := 1; END_IF;
    L_Buffer_Count := L_Buffer_Count - 1;
    L_Has_Command_To_Process := TRUE;
END_IF;

// 3. Обработка команды
IF L_Has_Command_To_Process THEN
    // Проверка IP-адреса источника
    L_IP_Allowed := FALSE;
    IF L_Process_Command.source_ip = '' THEN
        L_IP_Allowed := TRUE; // Если IP не передан, пропускаем (для обратной совместимости или локальных вызовов)
    ELSE
        FOR L_i := 1 TO GVL_CONSTANTS.C_MAX_ALLOWED_IPS DO
            IF VI_Allowed_IPs[L_i] = L_Process_Command.source_ip THEN
                L_IP_Allowed := TRUE;
                EXIT;
            END_IF;
        END_FOR;
    END_IF;
    
    IF NOT L_IP_Allowed THEN
        VO_HMI_Status_Message := 'Gateway: Ошибка безопасности (Неизвестный IP)';
        RETURN;
    END_IF;

    // Проверка целостности данных (CRC32)
    // Размер данных для расчета CRC: размер структуры минус размер самого поля crc32
    L_Command_Size := SIZEOF(L_Process_Command) - SIZEOF(L_Process_Command.crc32);
    L_Calculated_CRC := L_CRC_Calc.Calculate(ADR(L_Process_Command), L_Command_Size);
    
    IF L_Calculated_CRC = L_Process_Command.crc32 THEN
        L_Deduplicator(
            VI_Command_ID := L_Process_Command.command_id,
            VI_Command_Type := L_Process_Command.command_type,
            VI_Command_Value := L_Process_Command.target_value,
            VI_System_Time_MS := VI_System_Time_MS
        );
        
        IF L_Deduplicator.VO_Is_New_Command THEN
            CASE L_Process_Command.command_type OF
        E_Gateway_Command_Type.CMD_SET_SCENARIO: // Управление сценариями
            VO_Set_Scenario_Req := TRUE;
            VO_Target_Scenario := L_Process_Command.target_scenario;
            VO_HMI_Status_Message := 'Gateway: Сценарий изменен';
        E_Gateway_Command_Type.CMD_SET_LIGHT: // Управление освещением
            IF (L_Process_Command.target_zone >= 1) AND (L_Process_Command.target_zone <= GVL_CONSTANTS.C_MAX_LIGHTING_ZONES) THEN
                VO_Lighting_Override[L_Process_Command.target_zone] := TO_BYTE(L_Process_Command.target_value);
                VO_HMI_Status_Message := 'Gateway: Команда освещения принята';
            END_IF;
        E_Gateway_Command_Type.CMD_SET_BLINDS: // Управление шторами
            IF (L_Process_Command.target_zone >= 1) AND (L_Process_Command.target_zone <= GVL_CONSTANTS.C_MAX_BLINDS) THEN
                VO_Blinds_Override[L_Process_Command.target_zone] := TO_BYTE(L_Process_Command.target_value);
                VO_HMI_Status_Message := 'Gateway: Команда штор принята';
            END_IF;
        E_Gateway_Command_Type.CMD_SET_SOCKET: // Розетки
            IF (L_Process_Command.target_zone >= 1) AND (L_Process_Command.target_zone <= GVL_CONSTANTS.C_MAX_SOCKETS) THEN
                VO_Socket_Override[L_Process_Command.target_zone] := L_Process_Command.target_on_off;
                VO_HMI_Status_Message := 'Gateway: Команда розетки принята';
            END_IF;
        E_Gateway_Command_Type.CMD_SET_SECURITY: // Охрана
            IF L_Process_Command.target_armed THEN
                VO_Arm_Req := TRUE;
            ELSE
                VO_Disarm_Req := TRUE;
            END_IF;
            VO_PIN_Code := L_Process_Command.target_pin;
            VO_2FA_Code_In := L_Process_Command.target_2fa_code;
            VO_HMI_Status_Message := 'Gateway: Запрос охраны принят';
        E_Gateway_Command_Type.CMD_SET_TEMP: // Управление температурой
            IF (L_Process_Command.target_zone >= 1) AND (L_Process_Command.target_zone <= GVL_CONSTANTS.C_MAX_LIGHTING_ZONES) THEN
                VO_Set_Temp_Req := TRUE;
                VO_Target_Zone := L_Process_Command.target_zone;
                VO_Target_Temp := L_Process_Command.target_value;
                VO_HMI_Status_Message := 'Gateway: Уставка температуры изменена';
            END_IF;
        E_Gateway_Command_Type.CMD_SET_VENT: // Управление вентиляцией
            // Пример: изменение скорости притока
            VO_Set_Vent_Req := TRUE;
            VO_Target_Vent_Speed := TO_BYTE(L_Process_Command.target_value);
            VO_HMI_Status_Message := 'Gateway: Уставка вентиляции изменена';
        E_Gateway_Command_Type.CMD_TELEGRAM_MSG: // Отправка сообщения в Telegram
            VO_Telegram_Msg := L_Process_Command.telegram_msg;
            VO_Send_Telegram := TRUE;
            VO_HMI_Status_Message := 'Gateway: Сообщение Telegram отправлено';
        E_Gateway_Command_Type.CMD_SYNC_TIME: // Синхронизация времени
            VO_Sync_Time_Req := TRUE;
            VO_New_Time_MS := TO_UDINT(L_Process_Command.target_value);
            VO_HMI_Status_Message := 'Gateway: Время синхронизировано';
        E_Gateway_Command_Type.CMD_ACK_ALARM: // Квитирование тревоги
            VO_Reset_Errors_Req := TRUE;
            VO_HMI_Status_Message := 'Gateway: Тревоги квитированы';
        E_Gateway_Command_Type.CMD_SET_CONFIG: // Обновление конфигурации
            VO_Set_Config_Req := TRUE;
            VO_HMI_Status_Message := 'Gateway: Запрос обновления конфигурации';
        END_CASE;
    END_IF;
ELSE
    VO_HMI_Status_Message := 'Gateway: Ошибка CRC команды';
END_IF;
END_IF;
// >>> BULK_SYNC_ANCHOR: FB_Gateway_Interface <<<

          
END_FUNCTION_BLOCK

FUNCTION_BLOCK FB_Heating_System_Manager
  VAR_INPUT
    VI_Maintenance_Zones : ARRAY[1..16] OF ST_Component_Maintenance;
    VI_Maintenance_Manifolds : ARRAY[1..5] OF ST_Component_Maintenance;
    VI_System_Time_MS : UDINT;
    VI_IsActivePLC : BOOL;
    VI_Outdoor_Temp : REAL;
    VI_Floor_Temps : ARRAY[1..16] OF REAL;
    VI_Room_Temps : ARRAY[1..16] OF REAL;
    VI_Config : ST_Heating_Config;
    VI_Manifold_Pressures : ARRAY[1..5] OF REAL;
    VI_Manifold_Currents : ARRAY[1..5] OF REAL;
    VI_Manifold_Temps_Supply : ARRAY[1..5] OF REAL;
    VI_Manifold_Temps_Return : ARRAY[1..5] OF REAL;
    VI_Boiler_Flame_Status : ARRAY[1..2] OF BOOL;
  END_VAR
  VAR_OUTPUT
    VO_Manifold_Valves : ARRAY[1..5] OF REAL;  (* 0-100% *)
    VO_Manifold_Pumps : ARRAY[1..5] OF BOOL;
    VO_Zone_Valves : ARRAY[1..16] OF BOOL;
    VO_Boiler_Enable : ARRAY[1..2] OF BOOL;
    VO_Boiler_Setpoint : ARRAY[1..2] OF REAL;  (* OpenTherm Setpoint *)
    VO_Status : ARRAY[1..5] OF ST_Manifold_Status;
    VO_Boiler_Status : ARRAY[1..2] OF ST_Boiler_Status;
  END_VAR
  VAR
    L_PID_Valves : ARRAY[1..5] OF FB_PID_Controller;
    L_Last_Boiler_Rotation : UDINT;
    L_Lead_Boiler : BYTE := 1;
    L_i : INT;
    L_Target_Supply_Temp : REAL;
    L_Demand_Power : REAL;
    L_Any_Zone_Active : ARRAY[1..5] OF BOOL;
    L_Overheat_Timer : ARRAY[1..16] OF TON;  (* ТЗ 2.5: Задержка перегрева *)
    L_Pump_Run_Timer : ARRAY[1..5] OF TON;  (* ТЗ 2.6: Диагностика *)
    L_Pump_Pause_Timer : ARRAY[1..5] OF TON;
    L_Pump_In_Pause : ARRAY[1..5] OF BOOL;
    L_Last_Scan_Time : UDINT;  (* ТЗ 2.8: Учет наработки *)
    L_Lifespan_S : REAL := 180000000;  (* 50,000 hours in seconds *)
  END_VAR

            // ========================================
// Heating policy layer (phase2)
// ========================================
L_Policy_Normal := (VI_System_Mode = E_System_Operating_Mode.MODE_NORMAL);
L_Policy_Safe_Stop := (VI_System_Mode = E_System_Operating_Mode.MODE_SAFE_STOP);
L_Policy_Degraded := (VI_System_Mode = E_System_Operating_Mode.MODE_DEGRADED);
L_Policy_Freeze_Protection := (VI_System_Mode = E_System_Operating_Mode.MODE_FREEZE_PROTECTION);

// ========================================
// Heating freeze policy activation
// ========================================
IF L_Policy_Freeze_Protection THEN
    L_Freeze_Mode_Active := TRUE;
END_IF;

// 0. Агрегация деградации для system mode
GVL_STATE.G_Heating_IO_Fault := FALSE;
GVL_STATE.G_Heating_Sensor_Fault := FALSE;
GVL_STATE.G_Heating_Subsystem_Degraded := FALSE;
L_Any_Sensor_Error := FALSE;
L_Any_Subsystem_Degraded := FALSE;
L_Heating_V2_Shadow_Diff_Found := FALSE;
L_Heating_V2_Switch_Enabled := TRUE;
L_Heating_V2_Path_Ready := FALSE;
L_Heating_Using_Legacy_Fallback := TRUE;

// 0. Аварийный стоп от подсистемы безопасности
VO_Backup_Circulation_Pump := FALSE;
VO_Electric_Heater_Enable := FALSE;
VO_Freeze_Risk_Status := FALSE;

IF VI_Gas_Safety_Stop THEN
    L_Freeze_Mode_Active := (VI_Outdoor_Temp < -5.0);
    FOR L_i := 1 TO GVL_CONSTANTS.C_MAX_HEATING_CIRCUITS DO
        IF VI_Floor_Temps[L_i] < 7.0 THEN
            L_Freeze_Mode_Active := TRUE;
        END_IF;
        VO_Zone_Valves[L_i] := FALSE;
    END_FOR;

    FOR L_i := 1 TO GVL_CONSTANTS.C_MAX_MANIFOLDS DO
        VO_Manifold_Pumps[L_i] := FALSE;
        VO_Manifold_Valves[L_i] := 0.0;
    END_FOR;

    FOR L_i := 1 TO GVL_CONSTANTS.C_MAX_BOILERS DO
        VO_Boiler_OT_Enable[L_i] := FALSE;
        VO_Boiler_OT_Setpoint[L_i] := 0.0;
        VO_Boiler_Status[L_i].Warning := FALSE;
        VO_Boiler_Status[L_i].Error := TRUE;
    END_FOR;

    IF L_Freeze_Mode_Active THEN
        VO_Backup_Circulation_Pump := TRUE;
        L_Freeze_Target_Supply := LIMIT(20.0, VI_Config.Freeze_Threshold + 2.0, 35.0);
        L_Min_Supply_Temp := 1000.0;
        FOR L_i := 1 TO GVL_CONSTANTS.C_MAX_MANIFOLDS DO
            IF VI_Manifold_Temps_Supply[L_i] < L_Min_Supply_Temp THEN
                L_Min_Supply_Temp := VI_Manifold_Temps_Supply[L_i];
            END_IF;
        END_FOR;
        IF L_Min_Supply_Temp > 900.0 THEN
            L_Min_Supply_Temp := 0.0;
        END_IF;

        IF L_Min_Supply_Temp < (L_Freeze_Target_Supply - 1.0) THEN
            VO_Electric_Heater_Enable := TRUE;
        ELSIF L_Min_Supply_Temp > (L_Freeze_Target_Supply + 1.0) THEN
            VO_Electric_Heater_Enable := FALSE;
        END_IF;

        // При защёлкнутой газовой аварии оператор должен видеть, что система живёт в деградированном anti-freeze режиме.
        VO_Freeze_Risk_Status := TRUE;
    END_IF;

    RETURN;
END_IF;

IF VI_Emergency_Stop OR L_Policy_Safe_Stop THEN
    FOR L_i := 1 TO GVL_CONSTANTS.C_MAX_HEATING_CIRCUITS DO
        VO_Zone_Valves[L_i] := FALSE;
    END_FOR;

    FOR L_i := 1 TO GVL_CONSTANTS.C_MAX_MANIFOLDS DO
        VO_Manifold_Pumps[L_i] := FALSE;
        VO_Manifold_Valves[L_i] := 0.0;
    END_FOR;

    FOR L_i := 1 TO GVL_CONSTANTS.C_MAX_BOILERS DO
        VO_Boiler_OT_Enable[L_i] := FALSE;
        VO_Boiler_OT_Setpoint[L_i] := 0.0;
        VO_Boiler_Status[L_i].Warning := FALSE;
        VO_Boiler_Status[L_i].Error := TRUE;
    END_FOR;

    RETURN;
END_IF;

// 1. Проверка связи с модулями ввода-вывода (ТЗ 2.0)
L_IO_Failsafe_Active := FALSE;
FOR L_i := 1 TO GVL_CONSTANTS.C_MAX_MODULES DO
    IF NOT VI_IO_Modules_Online[L_i] THEN
        L_IO_Failsafe_Active := TRUE;
        GVL_STATE.G_Heating_IO_Fault := TRUE;
GVL_STATE.G_Heating_Subsystem_Degraded := TRUE;
        EXIT;
    END_IF;
END_FOR;

IF L_IO_Failsafe_Active THEN
    // Fail-safe: закрываем зональные клапаны, чтобы не разгонять неконтролируемые контуры,
    // но при риске замерзания сохраняем минимальную циркуляцию и минимальную теплогенерацию.
    L_Freeze_Mode_Active := (VI_Outdoor_Temp < -5.0);

    FOR L_j := 1 TO GVL_CONSTANTS.C_MAX_HEATING_CIRCUITS DO
        IF VI_Floor_Temps[L_j] < 7.0 THEN
            L_Freeze_Mode_Active := TRUE;
        END_IF;
        VO_Zone_Valves[L_j] := FALSE;
    END_FOR;

    IF L_Freeze_Mode_Active THEN
        L_Freeze_Target_Supply := LIMIT(20.0, VI_Config.Freeze_Threshold + 2.0, 35.0);
    ELSE
        L_Freeze_Target_Supply := 0.0;
    END_IF;

    FOR L_j := 1 TO GVL_CONSTANTS.C_MAX_MANIFOLDS DO
        IF L_Freeze_Mode_Active THEN
            VO_Manifold_Pumps[L_j] := TRUE;
            VO_Manifold_Valves[L_j] := 35.0;
        ELSE
            VO_Manifold_Pumps[L_j] := FALSE;
            VO_Manifold_Valves[L_j] := 0.0;
        END_IF;
    END_FOR;

    // В аварийном I/O режиме напрямую формируем только legacy request-мirror.
    // Реальные физические команды всё равно будут интерпретированы transport-слоем выше по архитектуре.
    FOR L_j := 1 TO GVL_CONSTANTS.C_MAX_BOILERS DO
        VO_Boiler_OT_Enable[L_j] := FALSE;
        VO_Boiler_OT_Setpoint[L_j] := 0.0;
    END_FOR;

    IF L_Freeze_Mode_Active THEN
        // В fail-safe используем только ведущий аварийный вариант: котёл №1 на минимальной уставке.
        IF VI_Boiler_OT_Online[1] AND NOT VI_Boiler_Error_Status[1] THEN
            VO_Boiler_OT_Enable[1] := TRUE;
            VO_Boiler_OT_Setpoint[1] := L_Freeze_Target_Supply;
        END_IF;
    END_IF;

    RETURN;
END_IF;

// 2. Расчет целевой температуры подачи теплоносителя (Погодозависимая автоматика ТЗ 2.3)
L_Target_Supply_Temp := 35.0; // Базовая уставка
IF VI_Config.Weather_Comp_Enabled AND VI_Outdoor_Temp < 15.0 THEN
    // Коррекция по уличному датчику с использованием коэффициента кривой
    L_Target_Supply_Temp := L_Target_Supply_Temp + (15.0 - VI_Outdoor_Temp) * VI_Config.Weather_Coef;
END_IF;
L_Target_Supply_Temp := LIMIT(20.0, L_Target_Supply_Temp, 45.0); // Ограничение диапазона для теплого пола

IF L_Policy_Degraded THEN
    IF L_Target_Supply_Temp > 35.0 THEN
        L_Target_Supply_Temp := 35.0;
    END_IF;
END_IF;

// Плавный переход уставки по сценарию
IF VI_Current_Scenario >= 1 AND VI_Current_Scenario <= GVL_CONSTANTS.C_MAX_SCENARIOS THEN
    L_Target_Scenario_Adjust := VI_Scenario_Configs[VI_Current_Scenario].floor_heating_adjust_celsius;
ELSE
    L_Target_Scenario_Adjust := 0.0;
END_IF;

IF VI_Current_Scenario <> L_Prev_Scenario THEN
    L_Transition_Temp(
        VI_System_Time := VI_System_Time_MS,
        VI_Start_Time := VI_System_Time_MS,
        VI_Duration := 300000, // 5 минут на плавное изменение температуры
        VI_Start_Value := L_Scenario_Adjust,
        VI_End_Value := L_Target_Scenario_Adjust
    );
    L_Prev_Scenario := VI_Current_Scenario;
ELSE
    L_Transition_Temp(
        VI_System_Time := VI_System_Time_MS,
        VI_Start_Time := L_Transition_Temp.VI_Start_Time,
        VI_Duration := L_Transition_Temp.VI_Duration,
        VI_Start_Value := L_Transition_Temp.VI_Start_Value,
        VI_End_Value := L_Target_Scenario_Adjust
    );
END_IF;
L_Scenario_Adjust := L_Transition_Temp.VO_Current_Value;

// ТЗ 2.4: Защита от замерзания по температуре пола < 7°C или наружной < -5°C
L_Freeze_Mode_Active := L_Policy_Freeze_Protection OR (VI_Outdoor_Temp < -5.0);
IF NOT L_Freeze_Mode_Active THEN
    FOR L_i := 1 TO GVL_CONSTANTS.C_MAX_HEATING_CIRCUITS DO
        IF VI_Floor_Temps[L_i] < 7.0 THEN
            L_Freeze_Mode_Active := TRUE;
            EXIT;
        END_IF;
    END_FOR;
END_IF;

IF L_Freeze_Mode_Active THEN
    L_Freeze_Target_Supply := LIMIT(20.0, VI_Config.Freeze_Threshold + 2.0, 45.0);
    IF L_Target_Supply_Temp < L_Freeze_Target_Supply THEN
        L_Target_Supply_Temp := L_Freeze_Target_Supply;
    END_IF;
END_IF;

// 2. Индивидуальное управление зонами отопления (ТЗ 1.1, 2.5)
FOR L_i := 1 TO GVL_CONSTANTS.C_MAX_HEATING_CIRCUITS DO
    fbFloorTempValidator[L_i](
        VI_Value := VI_Floor_Temps[L_i],
        VI_Min_Valid := -40.0,
        VI_Max_Valid := 120.0,
        VI_Fallback_Mode := 0
    );
    
    L_Climate_Zone_ID := VI_Zone_Configs[L_i].zone;
    IF L_Climate_Zone_ID >= 1 AND L_Climate_Zone_ID <= GVL_CONSTANTS.C_MAX_CLIMATE_ZONES THEN
        fbRoomTempValidator[L_Climate_Zone_ID](
        VI_Value := VI_Room_Temps[L_Climate_Zone_ID],
        VI_Min_Valid := -40.0,
        VI_Max_Valid := 120.0,
        VI_Fallback_Mode := 0
        );
    END_IF;

    // Контроль перегрева стяжки (защита напольного покрытия)
    L_Overheat_Timer[L_i](IN := fbFloorTempValidator[L_i].VO_Value > VI_Config.Overheat_Threshold, PT := T#60s, VI_System_Time_MS := VI_System_Time_MS);
    
    // Выбор датчика температуры с автоматическим переключением при неисправности
    L_Current_Temp := 0.0;
    L_Sensor_Error := FALSE;
    
    IF VI_Zone_Configs[L_i].control_type = 1 OR VI_Zone_Configs[L_i].control_type = 2 THEN
        // Основной: по воздуху
        IF NOT fbRoomTempValidator[L_Climate_Zone_ID].VO_Error THEN
            L_Current_Temp := fbRoomTempValidator[L_Climate_Zone_ID].VO_Value;
        ELSIF NOT fbFloorTempValidator[L_i].VO_Error THEN
            L_Current_Temp := fbFloorTempValidator[L_i].VO_Value; // Резервный: по полу
        ELSE
            L_Sensor_Error := TRUE;
        END_IF;
    ELSE
        // Основной: по полу
        IF NOT fbFloorTempValidator[L_i].VO_Error THEN
            L_Current_Temp := fbFloorTempValidator[L_i].VO_Value;
        ELSIF NOT fbRoomTempValidator[L_Climate_Zone_ID].VO_Error THEN
            L_Current_Temp := fbRoomTempValidator[L_Climate_Zone_ID].VO_Value; // Резервный: по воздуху
        ELSE
            L_Sensor_Error := TRUE;
        END_IF;
    END_IF;

    IF L_Sensor_Error THEN
        L_Any_Sensor_Error := TRUE;
        VO_Zone_Valves[L_i] := FALSE; // Безопасное состояние при ошибке обоих датчиков
    ELSE
        // ПИД-регулирование и ШИМ для каждой зоны
        // Применяем плавную корректировку уставки от сценария
        L_Zone_Config := VI_Zone_Configs[L_i];
        L_Zone_Config.design_temp := L_Zone_Config.design_temp + L_Scenario_Adjust;
        L_Floor_Controllers[L_i](
            VI_Current_Temp := L_Current_Temp,
            VI_Config := L_Zone_Config,
            VI_Tariff := VI_Tariff,
            VI_Current_Hour := VI_Current_Hour,
            VI_IsActivePLC := VI_IsActivePLC,
            VI_System_Time_MS := VI_System_Time_MS,
            VO_Valve_Bool => VO_Zone_Valves[L_i]
        );
    END_IF;
    
    // Принудительное закрытие клапана при перегреве пола (ТЗ 2.5)
    IF L_Overheat_Timer[L_i].Q THEN
        VO_Zone_Valves[L_i] := FALSE;
    END_IF;
    
    // Обработка действий от Rule Engine (ТЗ 13.0)
    FOR L_j := 1 TO GVL_CONSTANTS.C_MAX_RULES DO
        IF VI_Rule_Actions[L_j].Active AND VI_Rule_Actions[L_j].Target_ID = L_i THEN
            IF VI_Rule_Actions[L_j].Action_Type = E_Rule_Action_Type.ACTION_SET_FLOOR_HEATING THEN
                VO_Zone_Valves[L_i] := (VI_Rule_Actions[L_j].Value > 0.5);
            END_IF;
        END_IF;
    END_FOR;
END_FOR;

GVL_STATE.G_Heating_Sensor_Fault := L_Any_Sensor_Error;

// 3. Определение потребности в работе коллекторных насосов
FOR L_i := 1 TO GVL_CONSTANTS.C_MAX_MANIFOLDS DO
    L_Any_Zone_Active[L_i] := FALSE;
END_FOR;

FOR L_i := 1 TO GVL_CONSTANTS.C_MAX_HEATING_CIRCUITS DO
    IF VO_Zone_Valves[L_i] THEN
        L_j := VI_Zone_Configs[L_i].manifold_id;
        IF L_j >= 1 AND L_j <= GVL_CONSTANTS.C_MAX_MANIFOLDS THEN
            L_Any_Zone_Active[L_j] := TRUE;
        END_IF;
    END_IF;
END_FOR;

// 4. Управление смесительными узлами коллекторов (ТЗ 2.6, 12.2)
FOR L_i := 1 TO GVL_CONSTANTS.C_MAX_MANIFOLDS DO
    // ПИД-регулирование трехходового клапана для поддержания стабильной температуры подачи
    // Вызываем ПИД регулятор каждую секунду
    L_PID_Timer[L_i](IN := TRUE, PT := T#1s, VI_System_Time_MS := VI_System_Time_MS);
    IF L_PID_Timer[L_i].Q THEN
        L_PID_Timer[L_i](IN := FALSE, PT := T#1s, VI_System_Time_MS := VI_System_Time_MS); // Сброс таймера
        L_PID_Timer[L_i](IN := TRUE, PT := T#1s, VI_System_Time_MS := VI_System_Time_MS); // Перезапуск
        
        L_PID_Valves[L_i](
            VI_SetPoint := L_Target_Supply_Temp,
            VI_ProcessValue := VI_Manifold_Temps_Supply[L_i],
            VI_Kp := 2.0, VI_Tn := 120.0, VI_Tv := 0.0,
            VI_Y_Min := 0.0, VI_Y_Max := 100.0, VI_Cycle_Time_S := 1.0,
            VO_Output => VO_Manifold_Valves[L_i]
        );
    END_IF;

    // ТЗ 2.6: Реализация обязательной паузы насоса (защита от закисания и перегрева при 72ч работе)
    L_Pump_Run_Timer[L_i](IN := VO_Manifold_Pumps[L_i] AND NOT L_Pump_In_Pause[L_i], PT := T#72h, VI_System_Time_MS := VI_System_Time_MS);
    IF L_Pump_Run_Timer[L_i].Q THEN L_Pump_In_Pause[L_i] := TRUE; END_IF;
    
    L_Pump_Pause_Timer[L_i](IN := L_Pump_In_Pause[L_i], PT := T#1h, VI_System_Time_MS := VI_System_Time_MS);
    IF L_Pump_Pause_Timer[L_i].Q THEN L_Pump_In_Pause[L_i] := FALSE; END_IF;

    // Включение насоса при наличии запроса от зон и отсутствии сервисной паузы
    // Приоритет ГВС: если есть запрос от ГВС, отключаем насосы отопления и закрываем клапаны
    IF VI_DHW_Heating_Demand THEN
        VO_Manifold_Pumps[L_i] := FALSE;
        VO_Manifold_Valves[L_i] := 0.0; // Принудительно закрываем смесительный клапан
    ELSE
        VO_Manifold_Pumps[L_i] := VI_IsActivePLC AND L_Any_Zone_Active[L_i] AND NOT L_Pump_In_Pause[L_i];
    END_IF;

    // Защита от замерзания системы (ТЗ 2.4)
        IF L_Freeze_Mode_Active THEN
            VO_Manifold_Pumps[L_i] := TRUE;
            IF VO_Manifold_Valves[L_i] < 35.0 THEN
                VO_Manifold_Valves[L_i] := 35.0;
            END_IF;
        END_IF;

        // Сбор диагностических данных для визуализации на HMI
    VO_Status[L_i].Pump_On := VO_Manifold_Pumps[L_i];
    VO_Status[L_i].Pump_Current := VI_Manifold_Currents[L_i];
    VO_Status[L_i].Pressure := VI_Manifold_Pressures[L_i];
    VO_Status[L_i].Temp_Supply := VI_Manifold_Temps_Supply[L_i];
    VO_Status[L_i].Temp_Return := VI_Manifold_Temps_Return[L_i];
    VO_Status[L_i].Valve_Pos := VO_Manifold_Valves[L_i];
    
    // Предиктивная диагностика насоса
    L_Pump_Diag[L_i](
        VI_Current_Value := VI_Manifold_Currents[L_i],
        VI_Nominal_Value := 0.55, // Номинальный ток насоса по ТЗ: середина диапазона 0.3..0.8 А
        VI_Is_Running := VO_Manifold_Pumps[L_i],
        VI_Reset_Stats := FALSE,
        VI_System_Time_MS := VI_System_Time_MS,
        VIO_Health_Data := VO_Status[L_i].Health
    );
    
    // Автоматический контроль рабочих параметров (ток / давление / ΔT)
        IF VO_Manifold_Pumps[L_i] THEN
            L_Delta_T := VI_Manifold_Temps_Supply[L_i] - VI_Manifold_Temps_Return[L_i];

            // Контроль тока насоса:
            // Приоритет ошибок:
            // 1. Насос/ток
            // 2. Давление
            // 3. ΔT
            VO_Status[L_i].Error := FALSE;
            VO_Status[L_i].Error_ID := 0;

            IF VI_Manifold_Currents[L_i] <= 0.01 THEN
                VO_Status[L_i].Error := TRUE;
                VO_Status[L_i].Error_ID := GVL_CONFIG.ERR_PUMP_NO_CURRENT;
            ELSIF VI_Manifold_Currents[L_i] < 0.3 THEN
                VO_Status[L_i].Error := TRUE;
                VO_Status[L_i].Error_ID := GVL_CONFIG.ERR_PUMP_UNDERCURRENT;
            ELSIF VI_Manifold_Currents[L_i] > 1.5 THEN
                VO_Status[L_i].Error := TRUE;
                VO_Status[L_i].Error_ID := GVL_CONFIG.ERR_PUMP_OVERCURRENT;
            END_IF;

            // Проверка давления в системе (норма 1.5 - 2.5 бар)
            IF (NOT VO_Status[L_i].Error) AND (VI_Manifold_Pressures[L_i] < 1.5 OR VI_Manifold_Pressures[L_i] > 2.5) THEN
                VO_Status[L_i].Error := TRUE;
                VO_Status[L_i].Error_ID := GVL_CONFIG.ERR_PRESSURE_OUT_OF_RANGE;
            END_IF;

            // Проверка эффективности теплообмена (ΔT 5..10°C норма)
            IF NOT VO_Status[L_i].Error THEN
                IF L_Delta_T < 5.0 THEN
                    VO_Status[L_i].Error := TRUE;
                    VO_Status[L_i].Error_ID := GVL_CONFIG.ERR_DELTA_T_LOW;
                ELSIF L_Delta_T > 10.0 THEN
                    VO_Status[L_i].Error := TRUE;
                    VO_Status[L_i].Error_ID := GVL_CONFIG.ERR_DELTA_T_HIGH;
                END_IF;
            END_IF;
        END_IF;

        // ТЗ 12.2: Еженедельное тестирование запорной арматуры (предотвращение закисания)
    // Выполняется менеджером fbValveTestManager
END_FOR;

fbValveTestManager(
    VI_System_Time_MS := VI_System_Time_MS,
    VI_IsActivePLC := VI_IsActivePLC,
    VI_Valve_Currents := VI_Manifold_Currents,
    VI_Valve_End_Switches := VI_Manifold_End_Switches,
    VI_Config := VI_Valve_Test_Config
);

IF fbValveTestManager.VO_Test_Active THEN
    L_i := fbValveTestManager.VO_Current_Valve;
    IF L_i >= 1 AND L_i <= GVL_CONSTANTS.C_MAX_MANIFOLDS THEN
        IF fbValveTestManager.VO_Valve_Cmd[L_i] THEN
            VO_Manifold_Valves[L_i] := 100.0;
        ELSE
            VO_Manifold_Valves[L_i] := 0.0;
        END_IF;
        VO_Manifold_Pumps[L_i] := FALSE; // Отключаем насос при тестировании клапана
    END_IF;
END_IF;

// 5. Управление каскадом котлов (ТЗ 2.8, OpenTherm-only, без legacy mirror)
L_Demand_Power := 0.0;
FOR L_i := 1 TO GVL_CONSTANTS.C_MAX_MANIFOLDS DO
    IF VO_Manifold_Pumps[L_i] THEN
        L_Demand_Power := L_Demand_Power + VO_Manifold_Valves[L_i];
    END_IF;
END_FOR;

// В режиме антизамерзания обеспечиваем минимальный запрос тепла
IF L_Freeze_Mode_Active AND L_Demand_Power < 20.0 THEN
    L_Demand_Power := 20.0;
END_IF;

IF L_Policy_Degraded THEN
    IF L_Demand_Power > 60.0 THEN
        L_Demand_Power := 60.0;
    END_IF;
END_IF;

fbBoilerCascade(
    VI_Enable := VI_IsActivePLC AND ((L_Demand_Power > GVL_CONSTANTS.C_BOILER_CASCADE_MIN_DEMAND) OR L_Freeze_Mode_Active),
    VI_System_Time_MS := VI_System_Time_MS,
    VI_Boiler_Stop := FALSE,
    VI_DHW_Heating_Demand := VI_DHW_Heating_Demand,
    VI_DHW_Target_Temp := VI_DHW_Target_Temp,
    VI_Target_Supply_Temp := L_Target_Supply_Temp,
    VI_Demand_Power := L_Demand_Power,
    VI_Boiler_Flame_Status := VI_Boiler_Flame_Status,
    VI_Boiler_Error_Status := VI_Boiler_Error_Status,
    VI_Boiler_OT_Online := VI_Boiler_OT_Online,
    VI_Boiler_Modulation := VI_Boiler_Modulation,
    VO_Boiler_Enable => L_Boiler_Request_Enable,
    VO_Boiler_Setpoint => L_Boiler_Request_Setpoint,
    VO_Lead_Boiler => L_Lead_Boiler
);



// ========================================
// OT availability enforcement (no fallback)
// ========================================
FOR L_i := 1 TO GVL_CONSTANTS.C_MAX_BOILERS DO
    IF NOT VI_Boiler_OT_Online[L_i] OR VI_Boiler_Error_Status[L_i] THEN
        L_Boiler_Request_Enable[L_i] := FALSE;
        L_Boiler_Request_Setpoint[L_i] := 0.0;
    END_IF;
END_FOR;

fbBoilerOpenTherm(
    VI_Enable := L_Boiler_Request_Enable,
    VI_Setpoint := L_Boiler_Request_Setpoint,
    VI_OT_Online := VI_Boiler_OT_Online,
    VI_OT_Error := VI_Boiler_Error_Status,
    VO_OT_Enable => VO_Boiler_OT_Enable,
    VO_OT_Setpoint => VO_Boiler_OT_Setpoint,
    VO_OT_Command_Valid => L_Boiler_OT_Command_Valid
);


// ========================================
// Boiler status normalization
// ========================================
FOR L_i := 1 TO GVL_CONSTANTS.C_MAX_BOILERS DO
    // Базовый сброс диагностических флагов котла
    VO_Boiler_Status[L_i].Active := L_Boiler_Request_Enable[L_i];
    VO_Boiler_Status[L_i].Warning := FALSE;
    VO_Boiler_Status[L_i].Error := FALSE;

    // Приоритет причин:
    // 1. Нет канала OpenTherm
    // 2. Котёл вернул ошибку
    // 3. Есть запрос, но нет пламени
    IF NOT VI_Boiler_OT_Online[L_i] THEN
        VO_Boiler_Status[L_i].Error := TRUE;
        VO_Boiler_Status[L_i].Error_ID := GVL_CONFIG.ERR_BOILER_OFFLINE;
        L_Any_Subsystem_Degraded := TRUE;
    ELSIF VI_Boiler_Error_Status[L_i] THEN
        VO_Boiler_Status[L_i].Error := TRUE;
        VO_Boiler_Status[L_i].Error_ID := GVL_CONFIG.ERR_BOILER_GENERAL_FAULT;
        L_Any_Subsystem_Degraded := TRUE;
    ELSIF L_Boiler_Request_Enable[L_i] AND NOT VI_Boiler_Flame_Status[L_i] THEN
        VO_Boiler_Status[L_i].Warning := TRUE;
        VO_Boiler_Status[L_i].Error_ID := GVL_CONFIG.ERR_BOILER_NO_FLAME;
        L_Any_Subsystem_Degraded := TRUE;
    ELSE
        VO_Boiler_Status[L_i].Error_ID := 0;
    END_IF;
END_FOR;

// Расчет наработки и остаточного ресурса котлов (ТЗ 2.8)
IF NOT L_Scan_Time_Init THEN
    L_Last_Scan_Time := VI_System_Time_MS;
    L_Scan_Time_Init := TRUE;
END_IF;

L_Delta_MS := F_TimeDiff(VI_System_Time_MS, L_Last_Scan_Time);
IF L_Delta_MS > 1000 THEN
    L_Delta_MS := 1000; // Ограничение дельты для предотвращения скачков после перезагрузки
END_IF;

L_Last_Scan_Time := VI_System_Time_MS;

FOR L_i := 1 TO GVL_CONSTANTS.C_MAX_BOILERS DO
    VO_Boiler_Status[L_i].Work_Seconds := GVL_Retain.G_Boiler_Work_Seconds[L_i];
    
    IF VI_Boiler_Flame_Status[L_i] THEN
        GVL_Retain.G_Boiler_Accumulated_MS[L_i] := GVL_Retain.G_Boiler_Accumulated_MS[L_i] + L_Delta_MS;
        IF GVL_Retain.G_Boiler_Accumulated_MS[L_i] >= GVL_CONSTANTS.C_MS_IN_SECOND THEN
            GVL_Retain.G_Boiler_Work_Seconds[L_i] := GVL_Retain.G_Boiler_Work_Seconds[L_i] + (GVL_Retain.G_Boiler_Accumulated_MS[L_i] / 1000);
            GVL_Retain.G_Boiler_Accumulated_MS[L_i] := GVL_Retain.G_Boiler_Accumulated_MS[L_i] MOD 1000;
            
            // Защита от переполнения (сброс при достижении ~136 лет)
            IF GVL_Retain.G_Boiler_Work_Seconds[L_i] > 4000000000 THEN
                GVL_Retain.G_Boiler_Work_Seconds[L_i] := 0;
            END_IF;
            
            VO_Boiler_Status[L_i].Work_Seconds := GVL_Retain.G_Boiler_Work_Seconds[L_i];
        END_IF;
    END_IF;
    
    VO_Boiler_Status[L_i].Work_Hours := TO_REAL(VO_Boiler_Status[L_i].Work_Seconds) / 3600.0;
    
    L_Boiler_Life[L_i](
        VI_Runtime_Hours := TO_UDINT(VO_Boiler_Status[L_i].Work_Hours),
        VI_Start_Count := 0, // Не считаем пуски для котлов в этой версии
        VI_Nominal_Life := 50000 // 50,000 часов
    );
    VO_Boiler_Status[L_i].Resource_Percent := TO_REAL(L_Boiler_Life[L_i].VO_Remaining_Percent);
    VO_Boiler_Status[L_i].Running := VI_Boiler_Flame_Status[L_i];
END_FOR;
GVL_STATE.G_Heating_Subsystem_Degraded := L_Any_Subsystem_Degraded;

// ========================================
// Heating V2 shadow execution (phase2)
// ========================================
fbHeatingV2Staging(
    VI_Zone_ID := 1,
    VI_Enable := TRUE,
    VI_Target_Temp := 22.0,
    VI_Valve_Position_Setpoint := 50.0,
    VI_Pump_Enable := TRUE,

    VI_Is_Active := TRUE,
    VI_Room_Temp := 21.0,
    VI_Supply_Temp := 35.0,
    VI_Return_Temp := 30.0,
    VI_Valve_Position_Actual := 50.0,
    VI_Alarm_Active := FALSE,

    VO_Command_Shadow => L_Heating_V2_Command_Shadow,
    VO_State_Shadow => L_Heating_V2_State_Shadow
);

// Heating V2 shadow validation
IF ABS(VO_Manifold_Valves[1] - L_Heating_V2_Command_Shadow.Valve_Position_Setpoint) > 0.1 THEN
    L_Heating_V2_Shadow_Diff_Found := TRUE;
END_IF;
IF ABS(VI_Room_Temps[1] - L_Heating_V2_State_Shadow.Room_Temp) > 0.1 THEN
    L_Heating_V2_Shadow_Diff_Found := TRUE;
END_IF;
IF ABS(VI_Manifold_Temps_Supply[1] - L_Heating_V2_State_Shadow.Supply_Temp) > 0.1 THEN
    L_Heating_V2_Shadow_Diff_Found := TRUE;
END_IF;

// Guarded Heating V2 enable
IF L_Heating_V2_Switch_Enabled THEN
    IF NOT L_Heating_V2_Shadow_Diff_Found THEN
        L_Heating_V2_Path_Ready := TRUE;
        L_Heating_Using_Legacy_Fallback := FALSE;
    ELSE
        L_Heating_V2_Path_Ready := FALSE;
        L_Heating_Using_Legacy_Fallback := TRUE;
    END_IF;
ELSE
    L_Heating_V2_Path_Ready := FALSE;
    L_Heating_Using_Legacy_Fallback := TRUE;
END_IF;


END_FUNCTION_BLOCK
// >>> BULK_SYNC_ANCHOR: FB_Heating_System_Manager <<<

          
END_FUNCTION_BLOCK

FUNCTION_BLOCK FB_History_Manager
  VAR_INPUT
    VI_System_Time_MS : UDINT;
    VI_Write_Event : BOOL;
    VI_Event : ST_History_Record;
  END_VAR
  VAR_OUTPUT
    VO_Total_Events : UDINT;
  END_VAR
  VAR
    L_History_Buffer : ARRAY[1..100] OF ST_History_Record;
    L_Write_Idx : INT := 1;
  END_VAR

            IF VI_Write_Event AND NOT L_Prev_Write_Event THEN
    GVL_Retain.G_History_Buffer[GVL_Retain.G_History_Write_Idx] := VI_Event;
    GVL_Retain.G_History_Buffer[GVL_Retain.G_History_Write_Idx].timestamp_ms := VI_System_Time_MS;
    
    GVL_Retain.G_History_Write_Idx := (GVL_Retain.G_History_Write_Idx MOD GVL_CONSTANTS.C_MAX_HISTORY_RECORDS) + 1;
    GVL_Retain.G_History_Total_Events := GVL_Retain.G_History_Total_Events + 1;
END_IF;
L_Prev_Write_Event := VI_Write_Event;

VO_Total_Events := GVL_Retain.G_History_Total_Events;
// >>> BULK_SYNC_ANCHOR: FB_History_Manager <<<

          
END_FUNCTION_BLOCK

FUNCTION_BLOCK FB_Lifetime_Predictor
  VAR_INPUT
    VI_Runtime_Hours : UDINT;
    VI_Start_Count : UDINT;
    VI_Nominal_Life : UDINT := 10000;
  END_VAR
  VAR_OUTPUT
    VO_Remaining_Percent : BYTE;
    VO_Maintenance_Req : BOOL;
  END_VAR

            // Упрощенная модель износа
IF VI_Nominal_Life > 0 THEN
    VO_Remaining_Percent := TO_BYTE(100 - (VI_Runtime_Hours * 100 / VI_Nominal_Life));
ELSE
    VO_Remaining_Percent := 0;
END_IF;

VO_Maintenance_Req := (VO_Remaining_Percent < 10);

          
END_FUNCTION_BLOCK

FUNCTION_BLOCK FB_Lighting_Blinds_Manager
  VAR_INPUT
    VI_System_Time_MS : UDINT;
    VI_IsActivePLC : BOOL;
    VI_Current_Scenario : E_SCENARIO_TYPE;
    VI_Away_Level : BYTE;  (* 1-Short, 2-Medium, 3-Long *)
    VI_Simulation_Active : BOOL;
    VI_Manual_Light_Override : ARRAY[1..16] OF BYTE;  (* 0-100 *)
    VI_Manual_Blinds_Override : ARRAY[1..20] OF BYTE;  (* 0-100 *)
    VI_Simulation_Lights : ARRAY[1..16] OF BOOL;
    VI_Physical_Switches : ARRAY[1..16] OF BOOL;  (* ТЗ 1.0 *)
    VI_Motion_Sensors : ARRAY[1..16] OF BOOL;  (* ТЗ 2.0 *)
    VI_Maintenance : ARRAY[1..16] OF ST_Component_Maintenance;  (* ТЗ 6.0 *)
  END_VAR
  VAR_OUTPUT
    VO_Lighting_Levels : ARRAY[1..16] OF BYTE;
    VO_Blinds_Positions : ARRAY[1..20] OF BYTE;
    VO_Wet_Zone_Light_Active : ARRAY[1..4] OF BOOL;  (* Для вентиляции (ТЗ 4.0) *)
  END_VAR
  VAR
    L_i : INT;
    L_Base_Light : BYTE;
    L_Base_Blinds : BYTE;
    L_Light_States : ARRAY[1..16] OF BOOL;
    L_Prev_Switches : ARRAY[1..16] OF BOOL;
    L_Motion_Timers : ARRAY[1..16] OF TON;
  END_VAR

            IF NOT VI_IsActivePLC THEN RETURN; END_IF;

L_Lighting_V2_Shadow_Diff_Found := FALSE;
L_Blinds_V2_Shadow_Diff_Found := FALSE;
L_Blinds_V2_Switch_Enabled := TRUE;
L_Blinds_V2_Path_Ready := FALSE;
L_Blinds_Using_Legacy_Fallback := TRUE;
L_Lighting_V2_Switch_Enabled := TRUE;
L_Lighting_V2_Path_Ready := FALSE;
L_Lighting_Using_Legacy_Fallback := TRUE;

GVL_STATE.G_Lighting_IO_Fault := FALSE;
GVL_STATE.G_Lighting_Subsystem_Degraded := FALSE;

L_Effective_Scenario := VI_Current_Scenario;
L_Effective_Simulation_Active := VI_Simulation_Active;

CASE VI_System_Mode OF
    E_System_Operating_Mode.MODE_SAFE_STOP:
        FOR L_j := 1 TO GVL_CONSTANTS.C_MAX_LIGHTING_ZONES DO
            VO_Lighting_Levels[L_j] := 0;
        END_FOR;
        FOR L_j := 1 TO GVL_CONSTANTS.C_MAX_BLINDS DO
            VO_Blinds_Positions[L_j] := 100;
        END_FOR;
        FOR L_j := 1 TO GVL_CONSTANTS.C_MAX_WET_ZONES DO
            VO_Wet_Zone_Light_Active[L_j] := FALSE;
        END_FOR;
        RETURN;
    E_System_Operating_Mode.MODE_FREEZE_PROTECTION:
        L_Effective_Scenario := E_SCENARIO_TYPE.SCENARIO_NONE;
        L_Effective_Simulation_Active := FALSE;
    E_System_Operating_Mode.MODE_DEGRADED:
        L_Effective_Simulation_Active := FALSE;
END_CASE;

// Инициализация индекса мокрых зон
L_Wet_Zone_Idx := 1;
// Сброс массива мокрых зон
FOR L_i := 1 TO GVL_CONSTANTS.C_MAX_WET_ZONES DO
    VO_Wet_Zone_Light_Active[L_i] := FALSE;
END_FOR;

// Проверка связи с модулями ввода-вывода
FOR L_i := 1 TO GVL_CONSTANTS.C_MAX_MODULES DO
    IF NOT VI_IO_Modules_Online[L_i] THEN
        GVL_STATE.G_Lighting_IO_Fault := TRUE;
GVL_STATE.G_Lighting_Subsystem_Degraded := TRUE;
        // Переход в безопасное состояние при потере связи (свет выкл, шторы открыты для эвакуации)
        FOR L_j := 1 TO GVL_CONSTANTS.C_MAX_LIGHTING_ZONES DO
            VO_Lighting_Levels[L_j] := 0;
        END_FOR;
        FOR L_j := 1 TO GVL_CONSTANTS.C_MAX_BLINDS DO
            VO_Blinds_Positions[L_j] := 100;
        END_FOR;
        RETURN;
    END_IF;
END_FOR;

// 1. Определение целевых уровней по сценарию (ТЗ 7.1)
IF L_Effective_Scenario >= 1 AND L_Effective_Scenario <= GVL_CONSTANTS.C_MAX_SCENARIOS THEN
    L_Target_Base_Light := VI_Scenario_Configs[L_Effective_Scenario].lighting_level_base;
    L_Target_Base_Blinds := VI_Scenario_Configs[L_Effective_Scenario].blinds_position_percent;
ELSE
    L_Target_Base_Light := 100;
    L_Target_Base_Blinds := 100;
END_IF;

// Корректировка по астрономическому таймеру
IF VI_Is_Night AND L_Effective_Scenario <> E_SCENARIO_TYPE.SCENARIO_AWAY AND L_Effective_Scenario <> E_SCENARIO_TYPE.SCENARIO_SLEEP THEN
    L_Target_Base_Blinds := 0; // Закрывать шторы ночью
END_IF;

// Плавный переход при смене сценария
IF L_Effective_Scenario <> L_Prev_Scenario THEN
    L_Transition_Light(
        VI_System_Time := VI_System_Time_MS,
        VI_Start_Time := VI_System_Time_MS,
        VI_Duration := 5000, // 5 секунд на плавное изменение света
        VI_Start_Value := TO_REAL(L_Base_Light),
        VI_End_Value := TO_REAL(L_Target_Base_Light)
    );
    L_Transition_Blinds(
        VI_System_Time := VI_System_Time_MS,
        VI_Start_Time := VI_System_Time_MS,
        VI_Duration := 10000, // 10 секунд на плавное изменение штор
        VI_Start_Value := TO_REAL(L_Base_Blinds),
        VI_End_Value := TO_REAL(L_Target_Base_Blinds)
    );
    L_Prev_Scenario := L_Effective_Scenario;
ELSE
    L_Transition_Light(
        VI_System_Time := VI_System_Time_MS,
        VI_Start_Time := L_Transition_Light.VI_Start_Time,
        VI_Duration := L_Transition_Light.VI_Duration,
        VI_Start_Value := L_Transition_Light.VI_Start_Value,
        VI_End_Value := TO_REAL(L_Target_Base_Light)
    );
    L_Transition_Blinds(
        VI_System_Time := VI_System_Time_MS,
        VI_Start_Time := L_Transition_Blinds.VI_Start_Time,
        VI_Duration := L_Transition_Blinds.VI_Duration,
        VI_Start_Value := L_Transition_Blinds.VI_Start_Value,
        VI_End_Value := TO_REAL(L_Target_Base_Blinds)
    );
END_IF;

L_Base_Light := TO_BYTE(L_Transition_Light.VO_Current_Value);
L_Base_Blinds := TO_BYTE(L_Transition_Blinds.VO_Current_Value);

// 2. Управление освещением
FOR L_i := 1 TO GVL_CONSTANTS.C_MAX_LIGHTING_ZONES DO
    L_Rule_Light_Active := FALSE;
    L_Rule_Light_Val := 0;
    
